IF in > DatatypeLimits.MAX_VALUE_OF_ULINT_WHICH_CAN_BE_HELD_IN_A_UINT THEN
	RETURN;
END_IF

out := ULINT_TO_UINT(in);
TryConvert_ULINT_TO_UINT := TRUE;

END_FUNCTION

// mobject-converters/Converters/ULINT_TO_/TryConvert_ULINT_TO_UDINT
FUNCTION TryConvert_ULINT_TO_UDINT : BOOL
VAR_INPUT
	in : ULINT;
	out : REFERENCE TO UDINT;
END_VAR

IF in > DatatypeLimits.MAX_VALUE_OF_ULINT_WHICH_CAN_BE_HELD_IN_A_UDINT THEN
	RETURN;
END_IF

out := ULINT_TO_UDINT(in);
TryConvert_ULINT_TO_UDINT := TRUE;

END_FUNCTION

// mobject-converters/Converters/ULINT_TO_/TryConvert_ULINT_TO_ULINT
FUNCTION TryConvert_ULINT_TO_ULINT : BOOL
VAR_INPUT
	in : ULINT;
	out : REFERENCE TO ULINT;
END_VAR

out := in;
TryConvert_ULINT_TO_ULINT := TRUE;

END_FUNCTION

// mobject-converters/Converters/ULINT_TO_/TryConvert_ULINT_TO_REAL
FUNCTION TryConvert_ULINT_TO_REAL : BOOL
VAR_INPUT
	in : ULINT;
	out : REFERENCE TO REAL;
END_VAR

out := ULINT_TO_REAL(in);
TryConvert_ULINT_TO_REAL := TRUE;

END_FUNCTION

// mobject-converters/Converters/ULINT_TO_/TryConvert_ULINT_TO_LREAL
FUNCTION TryConvert_ULINT_TO_LREAL : BOOL
VAR_INPUT
	in : ULINT;
	out : REFERENCE TO LREAL;
END_VAR

out := ULINT_TO_LREAL(in);
TryConvert_ULINT_TO_LREAL := TRUE;

END_FUNCTION

// mobject-converters/Converters/ULINT_TO_/TryConvert_ULINT_TO_TIME
FUNCTION TryConvert_ULINT_TO_TIME : BOOL
VAR_INPUT
	in : ULINT;
	out : REFERENCE TO TIME;
END_VAR

IF in > DatatypeLimits.MAX_VALUE_OF_ULINT_WHICH_CAN_BE_HELD_IN_A_TIME THEN
	RETURN;
END_IF

out := ULINT_TO_TIME(in);
TryConvert_ULINT_TO_TIME := TRUE;

END_FUNCTION

// mobject-converters/Converters/ULINT_TO_/TryConvert_ULINT_TO_TOD
FUNCTION TryConvert_ULINT_TO_TOD : BOOL
VAR_INPUT
	in : ULINT;
	out : REFERENCE TO TOD;
END_VAR

IF in > DatatypeLimits.MAX_VALUE_OF_ULINT_WHICH_CAN_BE_HELD_IN_A_TOD THEN
	RETURN;
END_IF

out := ULINT_TO_TOD(in);
TryConvert_ULINT_TO_TOD := TRUE;

END_FUNCTION

// mobject-converters/Converters/ULINT_TO_/TryConvert_ULINT_TO_DT
FUNCTION TryConvert_ULINT_TO_DT : BOOL
VAR_INPUT
	in : ULINT;
	out : REFERENCE TO DT;
END_VAR

IF in > DatatypeLimits.MAX_VALUE_OF_ULINT_WHICH_CAN_BE_HELD_IN_A_DT THEN
	RETURN;
END_IF

out := ULINT_TO_DT(in);
TryConvert_ULINT_TO_DT := TRUE;

END_FUNCTION

// mobject-converters/Converters/ULINT_TO_/TryConvert_ULINT_TO_STRING
FUNCTION TryConvert_ULINT_TO_STRING : BOOL
VAR_INPUT
	in : ULINT;
	out : REFERENCE TO STRING;
END_VAR

out := ULINT_TO_STRING(in);
TryConvert_ULINT_TO_STRING := TRUE;

END_FUNCTION

// mobject-converters/Converters/USINT_TO_/TryConvert_USINT_TO_BOOL
FUNCTION TryConvert_USINT_TO_BOOL : BOOL
VAR_INPUT
	in : USINT;
	out : REFERENCE TO BOOL;
END_VAR

out := USINT_TO_BOOL(in);
TryConvert_USINT_TO_BOOL := TRUE;

END_FUNCTION

// mobject-converters/Converters/USINT_TO_/TryConvert_USINT_TO_BYTE
FUNCTION TryConvert_USINT_TO_BYTE : BOOL
VAR_INPUT
	in : USINT;
	out : REFERENCE TO BYTE;
END_VAR

out := USINT_TO_BYTE(in);
TryConvert_USINT_TO_BYTE := TRUE;

END_FUNCTION

// mobject-converters/Converters/USINT_TO_/TryConvert_USINT_TO_DATE
FUNCTION TryConvert_USINT_TO_DATE : BOOL
VAR_INPUT
	in : USINT;
	out : REFERENCE TO DATE;
END_VAR

out := USINT_TO_DATE(in);
TryConvert_USINT_TO_DATE := TRUE;

END_FUNCTION

// mobject-converters/Converters/USINT_TO_/TryConvert_USINT_TO_Destination
FUNCTION TryConvert_USINT_TO_Destination : BOOL
VAR_INPUT
	in : USINT;
	out : ANY;
END_VAR
VAR
	convertResult : BOOL := FALSE;
	convertAddress : PVOID;
	_BOOL : BOOL;
	_BYTE : BYTE;
	_WORD : WORD;
	_DWORD : DWORD;
	_LWORD : LWORD;
	_SINT : SINT;
	_INT : INT;
	_DINT : DINT;
	_LINT : LINT;
	_USINT : USINT;
	_UINT : UINT;
	_UDINT : UDINT;
	_ULINT : ULINT;
	_REAL : REAL;
	_LREAL : LREAL;
	_TIME : TIME;
	_TOD : TOD;
	_DATE : DATE;
	_DT : DT;
	_STRING : STRING;
END_VAR

CASE out.TypeClass OF
	__SYSTEM.TYPE_CLASS.TYPE_BOOL:
	
	convertResult := TryConvert_USINT_TO_BOOL(in, _BOOL);
	IF convertResult THEN
		convertAddress := ADR(_BOOL);
	END_IF
	
	__SYSTEM.TYPE_CLASS.TYPE_BYTE:
	
	convertResult := TryConvert_USINT_TO_BYTE(in, _BYTE);
	IF convertResult THEN
		convertAddress := ADR(_BYTE);
	END_IF
	
	__SYSTEM.TYPE_CLASS.TYPE_WORD:
	
	convertResult := TryConvert_USINT_TO_WORD(in, _WORD);
	IF convertResult THEN
		convertAddress := ADR(_WORD);
	END_IF
	
	__SYSTEM.TYPE_CLASS.TYPE_DWORD:
	
	convertResult := TryConvert_USINT_TO_DWORD(in, _DWORD);
	IF convertResult THEN
		convertAddress := ADR(_DWORD);
	END_IF
	
	__SYSTEM.TYPE_CLASS.TYPE_LWORD:
	
	convertResult := TryConvert_USINT_TO_LWORD(in, _LWORD);
	IF convertResult THEN
		convertAddress := ADR(_LWORD);
	END_IF
	
	__SYSTEM.TYPE_CLASS.TYPE_SINT:
	
	convertResult := TryConvert_USINT_TO_SINT(in, _SINT);
	IF convertResult THEN
		convertAddress := ADR(_SINT);
	END_IF
	
	__SYSTEM.TYPE_CLASS.TYPE_INT:
	
	convertResult := TryConvert_USINT_TO_INT(in, _INT);
	IF convertResult THEN
		convertAddress := ADR(_INT);
	END_IF
	
	__SYSTEM.TYPE_CLASS.TYPE_DINT:
	
	convertResult := TryConvert_USINT_TO_DINT(in, _DINT);
	IF convertResult THEN
		convertAddress := ADR(_DINT);
	END_IF
	
	__SYSTEM.TYPE_CLASS.TYPE_LINT:
	
	convertResult := TryConvert_USINT_TO_LINT(in, _LINT);
	IF convertResult THEN
		convertAddress := ADR(_LINT);
	END_IF
	
	__SYSTEM.TYPE_CLASS.TYPE_USINT:
	
	convertResult := TryConvert_USINT_TO_USINT(in, _USINT);
	IF convertResult THEN
		convertAddress := ADR(_USINT);
	END_IF
	
	__SYSTEM.TYPE_CLASS.TYPE_UINT:
	
	convertResult := TryConvert_USINT_TO_UINT(in, _UINT);
	IF convertResult THEN
		convertAddress := ADR(_UINT);
	END_IF
	
	__SYSTEM.TYPE_CLASS.TYPE_UDINT:
	
	convertResult := TryConvert_USINT_TO_UDINT(in, _UDINT);
	IF convertResult THEN
		convertAddress := ADR(_UDINT);
	END_IF
	
	__SYSTEM.TYPE_CLASS.TYPE_ULINT:
	
	convertResult := TryConvert_USINT_TO_ULINT(in, _ULINT);
	IF convertResult THEN
		convertAddress := ADR(_ULINT);
	END_IF
	
	__SYSTEM.TYPE_CLASS.TYPE_REAL:
	
	convertResult := TryConvert_USINT_TO_REAL(in, _REAL);
	IF convertResult THEN
		convertAddress := ADR(_REAL);
	END_IF
	
	__SYSTEM.TYPE_CLASS.TYPE_LREAL:
	
	convertResult := TryConvert_USINT_TO_LREAL(in, _LREAL);
	IF convertResult THEN
		convertAddress := ADR(_LREAL);
	END_IF
	
	__SYSTEM.TYPE_CLASS.TYPE_TIME:
	
	convertResult := TryConvert_USINT_TO_TIME(in, _TIME);
	IF convertResult THEN
		convertAddress := ADR(_TIME);
	END_IF
	
	__SYSTEM.TYPE_CLASS.TYPE_TIMEOFDAY:
	
	convertResult := TryConvert_USINT_TO_TOD(in, _TOD);
	IF convertResult THEN
		convertAddress := ADR(_TOD);
	END_IF
	
	__SYSTEM.TYPE_CLASS.TYPE_DATE:
	
	convertResult := TryConvert_USINT_TO_DATE(in, _DATE);
	IF convertResult THEN
		convertAddress := ADR(_DATE);
	END_IF
	
	__SYSTEM.TYPE_CLASS.TYPE_DATEANDTIME:
	
	convertResult := TryConvert_USINT_TO_DT(in, _DT);
	IF convertResult THEN
		convertAddress := ADR(_DT);
	END_IF
	
	__SYSTEM.TYPE_CLASS.TYPE_STRING:
	
	convertResult := TryConvert_USINT_TO_STRING(in, _STRING);
	IF convertResult THEN
		convertAddress := ADR(_STRING);
	END_IF
	
END_CASE

IF convertResult THEN
	memcpy(out.pValue,convertAddress,DINT_TO_UDINT(out.diSize));
END_IF

TryConvert_USINT_TO_Destination := convertResult;

END_FUNCTION

// mobject-converters/Converters/USINT_TO_/TryConvert_USINT_TO_WORD
FUNCTION TryConvert_USINT_TO_WORD : BOOL
VAR_INPUT
	in : USINT;
	out : REFERENCE TO WORD;
END_VAR

out := USINT_TO_WORD(in);
TryConvert_USINT_TO_WORD := TRUE;

END_FUNCTION

// mobject-converters/Converters/USINT_TO_/TryConvert_USINT_TO_DWORD
FUNCTION TryConvert_USINT_TO_DWORD : BOOL
VAR_INPUT
	in : USINT;
	out : REFERENCE TO DWORD;
END_VAR

out := USINT_TO_DWORD(in);
TryConvert_USINT_TO_DWORD := TRUE;

END_FUNCTION

// mobject-converters/Converters/USINT_TO_/TryConvert_USINT_TO_LWORD
FUNCTION TryConvert_USINT_TO_LWORD : BOOL
VAR_INPUT
	in : USINT;
	out : REFERENCE TO LWORD;
END_VAR

out := USINT_TO_LWORD(in);
TryConvert_USINT_TO_LWORD := TRUE;

END_FUNCTION

// mobject-converters/Converters/USINT_TO_/TryConvert_USINT_TO_SINT
FUNCTION TryConvert_USINT_TO_SINT : BOOL
VAR_INPUT
	in : USINT;
	out : REFERENCE TO SINT;
END_VAR

IF in > DatatypeLimits.MAX_VALUE_OF_USINT_WHICH_CAN_BE_HELD_IN_A_SINT THEN
	RETURN;
END_IF

out := USINT_TO_SINT(in);
TryConvert_USINT_TO_SINT := TRUE;

END_FUNCTION

// mobject-converters/Converters/USINT_TO_/TryConvert_USINT_TO_INT
FUNCTION TryConvert_USINT_TO_INT : BOOL
VAR_INPUT
	in : USINT;
	out : REFERENCE TO INT;
END_VAR

out := USINT_TO_INT(in);
TryConvert_USINT_TO_INT := TRUE;

END_FUNCTION

// mobject-converters/Converters/USINT_TO_/TryConvert_USINT_TO_DINT
FUNCTION TryConvert_USINT_TO_DINT : BOOL
VAR_INPUT
	in : USINT;
	out : REFERENCE TO DINT;
END_VAR

out := USINT_TO_DINT(in);
TryConvert_USINT_TO_DINT := TRUE;

END_FUNCTION

// mobject-converters/Converters/USINT_TO_/TryConvert_USINT_TO_LINT
FUNCTION TryConvert_USINT_TO_LINT : BOOL
VAR_INPUT
	in : USINT;
	out : REFERENCE TO LINT;
END_VAR

out := USINT_TO_LINT(in);
TryConvert_USINT_TO_LINT := TRUE;

END_FUNCTION

// mobject-converters/Converters/USINT_TO_/TryConvert_USINT_TO_USINT
FUNCTION TryConvert_USINT_TO_USINT : BOOL
VAR_INPUT
	in : USINT;
	out : REFERENCE TO USINT;
END_VAR

out := in;
TryConvert_USINT_TO_USINT := TRUE;

END_FUNCTION

// mobject-converters/Converters/USINT_TO_/TryConvert_USINT_TO_UINT
FUNCTION TryConvert_USINT_TO_UINT : BOOL
VAR_INPUT
	in : USINT;
	out : REFERENCE TO UINT;
END_VAR

out := USINT_TO_UINT(in);
TryConvert_USINT_TO_UINT := TRUE;

END_FUNCTION

// mobject-converters/Converters/USINT_TO_/TryConvert_USINT_TO_UDINT
FUNCTION TryConvert_USINT_TO_UDINT : BOOL
VAR_INPUT
	in : USINT;
	out : REFERENCE TO UDINT;
END_VAR

out := USINT_TO_UDINT(in);
TryConvert_USINT_TO_UDINT := TRUE;

END_FUNCTION

// mobject-converters/Converters/USINT_TO_/TryConvert_USINT_TO_ULINT
FUNCTION TryConvert_USINT_TO_ULINT : BOOL
VAR_INPUT
	in : USINT;
	out : REFERENCE TO ULINT;
END_VAR

out := USINT_TO_ULINT(in);
TryConvert_USINT_TO_ULINT := TRUE;

END_FUNCTION

// mobject-converters/Converters/USINT_TO_/TryConvert_USINT_TO_REAL
FUNCTION TryConvert_USINT_TO_REAL : BOOL
VAR_INPUT
	in : USINT;
	out : REFERENCE TO REAL;
END_VAR

out := USINT_TO_REAL(in);
TryConvert_USINT_TO_REAL := TRUE;

END_FUNCTION

// mobject-converters/Converters/USINT_TO_/TryConvert_USINT_TO_LREAL
FUNCTION TryConvert_USINT_TO_LREAL : BOOL
VAR_INPUT
	in : USINT;
	out : REFERENCE TO LREAL;
END_VAR

out := USINT_TO_LREAL(in);
TryConvert_USINT_TO_LREAL := TRUE;

END_FUNCTION

// mobject-converters/Converters/USINT_TO_/TryConvert_USINT_TO_TIME
FUNCTION TryConvert_USINT_TO_TIME : BOOL
VAR_INPUT
	in : USINT;
	out : REFERENCE TO TIME;
END_VAR

out := USINT_TO_TIME(in);
TryConvert_USINT_TO_TIME := TRUE;

END_FUNCTION

// mobject-converters/Converters/USINT_TO_/TryConvert_USINT_TO_TOD
FUNCTION TryConvert_USINT_TO_TOD : BOOL
VAR_INPUT
	in : USINT;
	out : REFERENCE TO TOD;
END_VAR

out := USINT_TO_TOD(in);
TryConvert_USINT_TO_TOD := TRUE;

END_FUNCTION

// mobject-converters/Converters/USINT_TO_/TryConvert_USINT_TO_DT
FUNCTION TryConvert_USINT_TO_DT : BOOL
VAR_INPUT
	in : USINT;
	out : REFERENCE TO DT;
END_VAR

out := USINT_TO_DT(in);
TryConvert_USINT_TO_DT := TRUE;

END_FUNCTION

// mobject-converters/Converters/USINT_TO_/TryConvert_USINT_TO_STRING
FUNCTION TryConvert_USINT_TO_STRING : BOOL
VAR_INPUT
	in : USINT;
	out : REFERENCE TO STRING;
END_VAR

out := USINT_TO_STRING(in);
TryConvert_USINT_TO_STRING := TRUE;

END_FUNCTION

// mobject-converters/Converters/WORD_TO_/TryConvert_WORD_TO_BOOL
FUNCTION TryConvert_WORD_TO_BOOL : BOOL
VAR_INPUT
	in : WORD;
	out : REFERENCE TO BOOL;
END_VAR

out := WORD_TO_BOOL(in);
TryConvert_WORD_TO_BOOL := TRUE;

END_FUNCTION

// mobject-converters/Converters/WORD_TO_/TryConvert_WORD_TO_BYTE
FUNCTION TryConvert_WORD_TO_BYTE : BOOL
VAR_INPUT
	in : WORD;
	out : REFERENCE TO BYTE;
END_VAR

IF in > DatatypeLimits.MAX_VALUE_OF_WORD_WHICH_CAN_BE_HELD_IN_A_BYTE THEN
	RETURN;
END_IF

out := WORD_TO_BYTE(in);
TryConvert_WORD_TO_BYTE := TRUE;

END_FUNCTION

// mobject-converters/Converters/WORD_TO_/TryConvert_WORD_TO_DATE
FUNCTION TryConvert_WORD_TO_DATE : BOOL
VAR_INPUT
	in : WORD;
	out : REFERENCE TO DATE;
END_VAR

out := WORD_TO_DATE(in);
TryConvert_WORD_TO_DATE := TRUE;

END_FUNCTION

// mobject-converters/Converters/WORD_TO_/TryConvert_WORD_TO_Destination
FUNCTION TryConvert_WORD_TO_Destination : BOOL
VAR_INPUT
	in : WORD;
	out : ANY;
END_VAR
VAR
	convertResult : BOOL := FALSE;
	convertAddress : PVOID;
	_BOOL : BOOL;
	_BYTE : BYTE;
	_WORD : WORD;
	_DWORD : DWORD;
	_LWORD : LWORD;
	_SINT : SINT;
	_INT : INT;
	_DINT : DINT;
	_LINT : LINT;
	_USINT : USINT;
	_UINT : UINT;
	_UDINT : UDINT;
	_ULINT : ULINT;
	_REAL : REAL;
	_LREAL : LREAL;
	_TIME : TIME;
	_TOD : TOD;
	_DATE : DATE;
	_DT : DT;
	_STRING : STRING;
END_VAR

CASE out.TypeClass OF
	__SYSTEM.TYPE_CLASS.TYPE_BOOL:
	
	convertResult := TryConvert_WORD_TO_BOOL(in, _BOOL);
	IF convertResult THEN
		convertAddress := ADR(_BOOL);
	END_IF
	
	__SYSTEM.TYPE_CLASS.TYPE_BYTE:
	
	convertResult := TryConvert_WORD_TO_BYTE(in, _BYTE);
	IF convertResult THEN
		convertAddress := ADR(_BYTE);
	END_IF
	
	__SYSTEM.TYPE_CLASS.TYPE_WORD:
	
	convertResult := TryConvert_WORD_TO_WORD(in, _WORD);
	IF convertResult THEN
		convertAddress := ADR(_WORD);
	END_IF
	
	__SYSTEM.TYPE_CLASS.TYPE_DWORD:
	
	convertResult := TryConvert_WORD_TO_DWORD(in, _DWORD);
	IF convertResult THEN
		convertAddress := ADR(_DWORD);
	END_IF
	
	__SYSTEM.TYPE_CLASS.TYPE_LWORD:
	
	convertResult := TryConvert_WORD_TO_LWORD(in, _LWORD);
	IF convertResult THEN
		convertAddress := ADR(_LWORD);
	END_IF
	
	__SYSTEM.TYPE_CLASS.TYPE_SINT:
	
	convertResult := TryConvert_WORD_TO_SINT(in, _SINT);
	IF convertResult THEN
		convertAddress := ADR(_SINT);
	END_IF
	
	__SYSTEM.TYPE_CLASS.TYPE_INT:
	
	convertResult := TryConvert_WORD_TO_INT(in, _INT);
	IF convertResult THEN
		convertAddress := ADR(_INT);
	END_IF
	
	__SYSTEM.TYPE_CLASS.TYPE_DINT:
	
	convertResult := TryConvert_WORD_TO_DINT(in, _DINT);
	IF convertResult THEN
		convertAddress := ADR(_DINT);
	END_IF
	
	__SYSTEM.TYPE_CLASS.TYPE_LINT:
	
	convertResult := TryConvert_WORD_TO_LINT(in, _LINT);
	IF convertResult THEN
		convertAddress := ADR(_LINT);
	END_IF
	
	__SYSTEM.TYPE_CLASS.TYPE_USINT:
	
	convertResult := TryConvert_WORD_TO_USINT(in, _USINT);
	IF convertResult THEN
		convertAddress := ADR(_USINT);
	END_IF
	
	__SYSTEM.TYPE_CLASS.TYPE_UINT:
	
	convertResult := TryConvert_WORD_TO_UINT(in, _UINT);
	IF convertResult THEN
		convertAddress := ADR(_UINT);
	END_IF
	
	__SYSTEM.TYPE_CLASS.TYPE_UDINT:
	
	convertResult := TryConvert_WORD_TO_UDINT(in, _UDINT);
	IF convertResult THEN
		convertAddress := ADR(_UDINT);
	END_IF
	
	__SYSTEM.TYPE_CLASS.TYPE_ULINT:
	
	convertResult := TryConvert_WORD_TO_ULINT(in, _ULINT);
	IF convertResult THEN
		convertAddress := ADR(_ULINT);
	END_IF
	
	__SYSTEM.TYPE_CLASS.TYPE_REAL:
	
	convertResult := TryConvert_WORD_TO_REAL(in, _REAL);
	IF convertResult THEN
		convertAddress := ADR(_REAL);
	END_IF
	
	__SYSTEM.TYPE_CLASS.TYPE_LREAL:
	
	convertResult := TryConvert_WORD_TO_LREAL(in, _LREAL);
	IF convertResult THEN
		convertAddress := ADR(_LREAL);
	END_IF
	
	__SYSTEM.TYPE_CLASS.TYPE_TIME:
	
	convertResult := TryConvert_WORD_TO_TIME(in, _TIME);
	IF convertResult THEN
		convertAddress := ADR(_TIME);
	END_IF
	
	__SYSTEM.TYPE_CLASS.TYPE_TIMEOFDAY:
	
	convertResult := TryConvert_WORD_TO_TOD(in, _TOD);
	IF convertResult THEN
		convertAddress := ADR(_TOD);
	END_IF
	
	__SYSTEM.TYPE_CLASS.TYPE_DATE:
	
	convertResult := TryConvert_WORD_TO_DATE(in, _DATE);
	IF convertResult THEN
		convertAddress := ADR(_DATE);
	END_IF
	
	__SYSTEM.TYPE_CLASS.TYPE_DATEANDTIME:
	
	convertResult := TryConvert_WORD_TO_DT(in, _DT);
	IF convertResult THEN
		convertAddress := ADR(_DT);
	END_IF
	
	__SYSTEM.TYPE_CLASS.TYPE_STRING:
	
	convertResult := TryConvert_WORD_TO_STRING(in, _STRING);
	IF convertResult THEN
		convertAddress := ADR(_STRING);
	END_IF
	
END_CASE

IF convertResult THEN
	memcpy(out.pValue,convertAddress,DINT_TO_UDINT(out.diSize));
END_IF

TryConvert_WORD_TO_Destination := convertResult;

END_FUNCTION

// mobject-converters/Converters/WORD_TO_/TryConvert_WORD_TO_WORD
FUNCTION TryConvert_WORD_TO_WORD : BOOL
VAR_INPUT
	in : WORD;
	out : REFERENCE TO WORD;
END_VAR

out := in;
TryConvert_WORD_TO_WORD := TRUE;

END_FUNCTION

// mobject-converters/Converters/WORD_TO_/TryConvert_WORD_TO_DWORD
FUNCTION TryConvert_WORD_TO_DWORD : BOOL
VAR_INPUT
	in : WORD;
	out : REFERENCE TO DWORD;
END_VAR

out := WORD_TO_DWORD(in);
TryConvert_WORD_TO_DWORD := TRUE;

END_FUNCTION

// mobject-converters/Converters/WORD_TO_/TryConvert_WORD_TO_LWORD
FUNCTION TryConvert_WORD_TO_LWORD : BOOL
VAR_INPUT
	in : WORD;
	out : REFERENCE TO LWORD;
END_VAR

out := WORD_TO_LWORD(in);
TryConvert_WORD_TO_LWORD := TRUE;

END_FUNCTION

// mobject-converters/Converters/WORD_TO_/TryConvert_WORD_TO_SINT
FUNCTION TryConvert_WORD_TO_SINT : BOOL
VAR_INPUT
	in : WORD;
	out : REFERENCE TO SINT;
END_VAR

IF in > DatatypeLimits.MAX_VALUE_OF_WORD_WHICH_CAN_BE_HELD_IN_A_SINT THEN
	RETURN;
END_IF

out := WORD_TO_SINT(in);
TryConvert_WORD_TO_SINT := TRUE;

END_FUNCTION

// mobject-converters/Converters/WORD_TO_/TryConvert_WORD_TO_INT
FUNCTION TryConvert_WORD_TO_INT : BOOL
VAR_INPUT
	in : WORD;
	out : REFERENCE TO INT;
END_VAR

IF in > DatatypeLimits.MAX_VALUE_OF_WORD_WHICH_CAN_BE_HELD_IN_A_INT THEN
	RETURN;
END_IF

out := WORD_TO_INT(in);
TryConvert_WORD_TO_INT := TRUE;

END_FUNCTION

// mobject-converters/Converters/WORD_TO_/TryConvert_WORD_TO_DINT
FUNCTION TryConvert_WORD_TO_DINT : BOOL
VAR_INPUT
	in : WORD;
	out : REFERENCE TO DINT;
END_VAR

out := WORD_TO_DINT(in);
TryConvert_WORD_TO_DINT := TRUE;

END_FUNCTION

// mobject-converters/Converters/WORD_TO_/TryConvert_WORD_TO_LINT
FUNCTION TryConvert_WORD_TO_LINT : BOOL
VAR_INPUT
	in : WORD;
	out : REFERENCE TO LINT;
END_VAR

out := WORD_TO_LINT(in);
TryConvert_WORD_TO_LINT := TRUE;

END_FUNCTION

// mobject-converters/Converters/WORD_TO_/TryConvert_WORD_TO_USINT
FUNCTION TryConvert_WORD_TO_USINT : BOOL
VAR_INPUT
	in : WORD;
	out : REFERENCE TO USINT;
END_VAR

IF in > DatatypeLimits.MAX_VALUE_OF_WORD_WHICH_CAN_BE_HELD_IN_A_USINT THEN
	RETURN;
END_IF

out := WORD_TO_USINT(in);
TryConvert_WORD_TO_USINT := TRUE;

END_FUNCTION

// mobject-converters/Converters/WORD_TO_/TryConvert_WORD_TO_UINT
FUNCTION TryConvert_WORD_TO_UINT : BOOL
VAR_INPUT
	in : WORD;
	out : REFERENCE TO UINT;
END_VAR

out := WORD_TO_UINT(in);
TryConvert_WORD_TO_UINT := TRUE;

END_FUNCTION

// mobject-converters/Converters/WORD_TO_/TryConvert_WORD_TO_UDINT
FUNCTION TryConvert_WORD_TO_UDINT : BOOL
VAR_INPUT
	in : WORD;
	out : REFERENCE TO UDINT;
END_VAR

out := WORD_TO_UDINT(in);
TryConvert_WORD_TO_UDINT := TRUE;

END_FUNCTION

// mobject-converters/Converters/WORD_TO_/TryConvert_WORD_TO_ULINT
FUNCTION TryConvert_WORD_TO_ULINT : BOOL
VAR_INPUT
	in : WORD;
	out : REFERENCE TO ULINT;
END_VAR

out := WORD_TO_ULINT(in);
TryConvert_WORD_TO_ULINT := TRUE;

END_FUNCTION

// mobject-converters/Converters/WORD_TO_/TryConvert_WORD_TO_REAL
FUNCTION TryConvert_WORD_TO_REAL : BOOL
VAR_INPUT
	in : WORD;
	out : REFERENCE TO REAL;
END_VAR

out := WORD_TO_REAL(in);
TryConvert_WORD_TO_REAL := TRUE;

END_FUNCTION

// mobject-converters/Converters/WORD_TO_/TryConvert_WORD_TO_LREAL
FUNCTION TryConvert_WORD_TO_LREAL : BOOL
VAR_INPUT
	in : WORD;
	out : REFERENCE TO LREAL;
END_VAR

out := WORD_TO_LREAL(in);
TryConvert_WORD_TO_LREAL := TRUE;

END_FUNCTION

// mobject-converters/Converters/WORD_TO_/TryConvert_WORD_TO_TIME
FUNCTION TryConvert_WORD_TO_TIME : BOOL
VAR_INPUT
	in : WORD;
	out : REFERENCE TO TIME;
END_VAR

out := WORD_TO_TIME(in);
TryConvert_WORD_TO_TIME := TRUE;

END_FUNCTION

// mobject-converters/Converters/WORD_TO_/TryConvert_WORD_TO_TOD
FUNCTION TryConvert_WORD_TO_TOD : BOOL
VAR_INPUT
	in : WORD;
	out : REFERENCE TO TOD;
END_VAR

out := WORD_TO_TOD(in);
TryConvert_WORD_TO_TOD := TRUE;

END_FUNCTION

// mobject-converters/Converters/WORD_TO_/TryConvert_WORD_TO_DT
FUNCTION TryConvert_WORD_TO_DT : BOOL
VAR_INPUT
	in : WORD;
	out : REFERENCE TO DT;
END_VAR

out := WORD_TO_DT(in);
TryConvert_WORD_TO_DT := TRUE;

END_FUNCTION

// mobject-converters/Converters/WORD_TO_/TryConvert_WORD_TO_STRING
FUNCTION TryConvert_WORD_TO_STRING : BOOL
VAR_INPUT
	in : WORD;
	out : REFERENCE TO STRING;
END_VAR

out := WORD_TO_STRING(in);
TryConvert_WORD_TO_STRING := TRUE;

END_FUNCTION

// mobject-converters/Converters/TryConvert_Source_TO_Destination
{attribute 'linkalways'} 
FUNCTION TryConvert_Source_TO_Destination : BOOL
VAR_INPUT
	in : ANY;
	out : ANY;
END_VAR
VAR
	_BOOL : BOOL;
	_BYTE : BYTE;
	_WORD : WORD;
	_DWORD : DWORD;
	_LWORD : LWORD;
	_SINT : SINT;
	_INT : INT;
	_DINT : DINT;
	_LINT : LINT;
	_USINT : USINT;
	_UINT : UINT;
	_UDINT : UDINT;
	_ULINT : ULINT;
	_REAL : REAL;
	_LREAL : LREAL;
	_TIME : TIME;
	_TOD : TOD;
	_DATE : DATE;
	_DT : DT;
	_STRING : STRING;
	convertResult : BOOL := FALSE;
END_VAR

CASE in.TypeClass OF

	__SYSTEM.TYPE_CLASS.TYPE_BOOL :
		memcpy(ADR(_BOOL),in.pValue,DINT_TO_UDINT(in.diSize));
		convertResult := TryConvert_BOOL_To_Destination(_BOOL, out);
		
	__SYSTEM.TYPE_CLASS.TYPE_BYTE :
		memcpy(ADR(_BYTE),in.pValue,DINT_TO_UDINT(in.diSize));
		convertResult := TryConvert_BYTE_To_Destination(_BYTE, out);
		
	__SYSTEM.TYPE_CLASS.TYPE_WORD :
		memcpy(ADR(_WORD),in.pValue,DINT_TO_UDINT(in.diSize));
		convertResult := TryConvert_WORD_To_Destination(_WORD, out);
		
	__SYSTEM.TYPE_CLASS.TYPE_DWORD :
		memcpy(ADR(_DWORD),in.pValue,DINT_TO_UDINT(in.diSize));
		convertResult := TryConvert_DWORD_To_Destination(_DWORD, out);
		
	__SYSTEM.TYPE_CLASS.TYPE_LWORD :
		memcpy(ADR(_LWORD),in.pValue,DINT_TO_UDINT(in.diSize));
		convertResult := TryConvert_LWORD_To_Destination(_LWORD, out);
		
	__SYSTEM.TYPE_CLASS.TYPE_SINT :
		memcpy(ADR(_SINT),in.pValue,DINT_TO_UDINT(in.diSize));
		convertResult := TryConvert_SINT_To_Destination(_SINT, out);
		
	__SYSTEM.TYPE_CLASS.TYPE_INT :
		memcpy(ADR(_INT),in.pValue,DINT_TO_UDINT(in.diSize));
		convertResult := TryConvert_INT_To_Destination(_INT, out);
		
	__SYSTEM.TYPE_CLASS.TYPE_DINT :
		memcpy(ADR(_DINT),in.pValue,DINT_TO_UDINT(in.diSize));
		convertResult := TryConvert_DINT_To_Destination(_DINT, out);
		
	__SYSTEM.TYPE_CLASS.TYPE_LINT :
		memcpy(ADR(_LINT),in.pValue,DINT_TO_UDINT(in.diSize));
		convertResult := TryConvert_LINT_To_Destination(_LINT, out);
		
	__SYSTEM.TYPE_CLASS.TYPE_USINT :
		memcpy(ADR(_USINT),in.pValue,DINT_TO_UDINT(in.diSize));
		convertResult := TryConvert_USINT_To_Destination(_USINT, out);
		
	__SYSTEM.TYPE_CLASS.TYPE_UINT :
		memcpy(ADR(_UINT),in.pValue,DINT_TO_UDINT(in.diSize));
		convertResult := TryConvert_UINT_To_Destination(_UINT, out);
		
	__SYSTEM.TYPE_CLASS.TYPE_UDINT :
		memcpy(ADR(_UDINT),in.pValue,DINT_TO_UDINT(in.diSize));
		convertResult := TryConvert_UDINT_To_Destination(_UDINT, out);
		
	__SYSTEM.TYPE_CLASS.TYPE_ULINT :
		memcpy(ADR(_ULINT),in.pValue,DINT_TO_UDINT(in.diSize));
		convertResult := TryConvert_ULINT_To_Destination(_ULINT, out);
		
	__SYSTEM.TYPE_CLASS.TYPE_REAL :
		memcpy(ADR(_REAL),in.pValue,DINT_TO_UDINT(in.diSize));
		convertResult := TryConvert_REAL_To_Destination(_REAL, out);
		
	__SYSTEM.TYPE_CLASS.TYPE_LREAL :
		memcpy(ADR(_LREAL),in.pValue,DINT_TO_UDINT(in.diSize));
		convertResult := TryConvert_LREAL_To_Destination(_LREAL, out);
		
	__SYSTEM.TYPE_CLASS.TYPE_TIME :
		memcpy(ADR(_TIME),in.pValue,DINT_TO_UDINT(in.diSize));
		convertResult := TryConvert_TIME_To_Destination(_TIME, out);
		
	__SYSTEM.TYPE_CLASS.TYPE_TIMEOFDAY :
		memcpy(ADR(_TOD),in.pValue,DINT_TO_UDINT(in.diSize));
		convertResult := TryConvert_TOD_To_Destination(_TOD, out);
		
	__SYSTEM.TYPE_CLASS.TYPE_DATE :
		memcpy(ADR(_DATE),in.pValue,DINT_TO_UDINT(in.diSize));
		convertResult := TryConvert_DATE_To_Destination(_DATE, out);
		
	__SYSTEM.TYPE_CLASS.TYPE_DATEANDTIME :
		memcpy(ADR(_DT),in.pValue,DINT_TO_UDINT(in.diSize));
		convertResult := TryConvert_DT_To_Destination(_DT, out);
		
	__SYSTEM.TYPE_CLASS.TYPE_STRING :
		memcpy(ADR(_STRING),in.pValue,DINT_TO_UDINT(in.diSize));
		convertResult := TryConvert_STRING_To_Destination(_STRING, out);
		
	END_CASE
TryConvert_Source_TO_Destination  := convertResult;

END_FUNCTION

// mobject-datatypes/_Internal/Datatype/AliasDatatypeBase
{attribute 'linkalways'} 
{attribute 'no_explicit_call' := 'This FB is a CLASS and must be accessed using methods or properties'}
{attribute 'enable_dynamic_creation'}
FUNCTION_BLOCK ABSTRACT AliasDatatypeBase EXTENDS UserDefinedDatatypeBase IMPLEMENTS I_AliasDatatype
VAR
	_baseDatatype : I_Datatype;
END_VAR

METHOD PROTECTED AddBaseDatatype
VAR_INPUT
	BaseType : I_Datatype;
END_VAR
_baseDatatype := BaseType;
END_METHOD

METHOD PROTECTED OnSerializeTypeWith
VAR_INPUT
	Serializer : I_Serializer;
END_VAR
SUPER^.OnSerializeTypeWith(Serializer);
Serializer.AddKey('baseDatatype');
_baseDatatype.SerializeTypeWith(Serializer);
END_METHOD

PROPERTY PUBLIC BaseDatatype : I_Datatype
GET
BaseDatatype := _baseDatatype;
END_GET
END_PROPERTY

METHOD PUBLIC SerializeWith
VAR_INPUT
	Serializer : I_Serializer;
END_VAR
_baseDatatype.SerializeWith(Serializer);
END_METHOD

METHOD TryDeserializeFrom : BOOL
VAR_INPUT
	Deserializer : I_Deserializer;
	Feedback : I_DeserializerFeedback;
END_VAR
TryDeserializeFrom := _baseDatatype.TryDeserializeFrom(Deserializer, Feedback);
END_METHOD

METHOD PUBLIC TryResolveAsAliasDatatype : BOOL
VAR_INPUT
	Destination : REFERENCE TO I_AliasDatatype;
END_VAR
Destination := THIS^;
TryResolveAsAliasDatatype := TRUE;
END_METHOD

PROPERTY PUBLIC TypeName : T_MAXSTRING
GET
TypeName := 'ALIAS';
END_GET
END_PROPERTY

END_FUNCTION_BLOCK

// mobject-datatypes/_Internal/Datatype/UserDefinedDatatypeBase
{attribute 'linkalways'} 
{attribute 'no_explicit_call' := 'This FB is a CLASS and must be accessed using methods or properties'}
{attribute 'enable_dynamic_creation'}
FUNCTION_BLOCK ABSTRACT UserDefinedDatatypeBase EXTENDS DatatypeBase IMPLEMENTS I_UserDefinedDatatype
VAR
END_VAR

METHOD PROTECTED OnSerializeTypeWith
VAR_INPUT
	Serializer : I_Serializer;
END_VAR
SUPER^.OnSerializeTypeWith(Serializer);
Serializer.AddKeyString('identifier',Identifier);
END_METHOD

PROPERTY PUBLIC ABSTRACT Identifier : T_MAXSTRING
GET
END_GET
END_PROPERTY

PROPERTY PUBLIC IsUserDefined : BOOL
GET
IsUserDefined := TRUE;
END_GET
END_PROPERTY

METHOD PUBLIC TryCopyFrom : BOOL
VAR_INPUT
	Source : I_Datatype;
END_VAR
VAR
	sourceAsUdt : I_UserDefinedDatatype;
END_VAR
IF NOT __QUERYINTERFACE(Source, sourceAsUdt) THEN
	RETURN;
END_IF

IF sourceAsUdt.Identifier <> Identifier THEN
	RETURN;
END_IF

TryCopyFrom := SUPER^.TryCopyFrom(Source);
END_METHOD

METHOD PUBLIC TryResolveAsUserDefinedDatatype : BOOL
VAR_INPUT
	Destination : REFERENCE TO I_UserDefinedDatatype;
END_VAR
Destination := THIS^;
TryResolveAsUserDefinedDatatype := TRUE;
END_METHOD

END_FUNCTION_BLOCK

// mobject-datatypes/_Internal/Datatype/ArrayDatatypeBase
{attribute 'linkalways'} 
{attribute 'no_explicit_call' := 'This FB is a CLASS and must be accessed using methods or properties'}
{attribute 'enable_dynamic_creation'}
FUNCTION_BLOCK ABSTRACT ArrayDatatypeBase EXTENDS UserDefinedDatatypeBase IMPLEMENTS I_ArrayDatatype
VAR
END_VAR

METHOD PRIVATE CreateEnumError : I_Error
VAR_INPUT
	Enum : T_MAXSTRING;
END_VAR
VAR
	pError : POINTER TO UnknownEnumerationError;
END_VAR
pError := __NEW(UnknownEnumerationError(EnumString := Enum));
CreateEnumError := pError^;
END_METHOD

METHOD PRIVATE SerializeBaseType
VAR_INPUT
	Serializer : I_Serializer;
END_VAR
IF BaseDatatype = 0 THEN
	RETURN;
END_IF

Serializer.AddKey('baseType');
BaseDatatype.SerializeTypeWith(Serializer);
END_METHOD

METHOD PROTECTED ABSTRACT OnSerializeArrayValues
VAR_INPUT
	Serializer : I_Serializer;
END_VAR
END_METHOD

METHOD PROTECTED OnSerializeTypeWith
VAR_INPUT
	Serializer : I_Serializer;
END_VAR
SUPER^.OnSerializeTypeWith(Serializer);
SerializeBaseType(Serializer);
END_METHOD

METHOD PROTECTED ABSTRACT TryDeserializeArrayValues : BOOL
VAR_INPUT
	Deserializer : I_Deserializer;
	Feedback : I_DeserializerFeedback;
END_VAR
END_METHOD

PROPERTY PUBLIC ABSTRACT BaseDatatype : I_Datatype
GET
END_GET
END_PROPERTY

METHOD PUBLIC ABSTRACT GetElementAsDatatypeByIndex : I_Datatype
VAR_INPUT
	Index : DINT;
END_VAR
END_METHOD

PROPERTY PUBLIC Identifier : T_MAXSTRING
GET
VAR
	baseTypeAsUdt : I_UserDefinedDatatype;
END_VAR
Identifier := Concat('ARRAY [', DINT_TO_STRING(LowerBound));
Identifier := Concat(Identifier,'..');
Identifier := Concat(Identifier, DINT_TO_STRING(UpperBound));
Identifier := Concat(Identifier, '] OF ');

IF BaseDatatype.TryResolveAsUserDefinedDatatype(baseTypeAsUdt) THEN
	Identifier := Concat(Identifier, baseTypeAsUdt.Identifier);
ELSE
	Identifier := Concat(Identifier, BaseDatatype.TypeName);
END_IF
END_GET
END_PROPERTY

PROPERTY PUBLIC Length : UDINT
GET
Length := ABS(UpperBound - LowerBound) + 1;
END_GET
END_PROPERTY

PROPERTY PUBLIC ABSTRACT LowerBound : DINT
GET
END_GET
END_PROPERTY

METHOD PUBLIC SerializeWith
VAR_INPUT
	Serializer : I_Serializer;
END_VAR
Serializer.StartArray();
OnSerializeArrayValues(Serializer);
Serializer.EndArray();
END_METHOD

METHOD TryDeserializeFrom : BOOL
VAR_INPUT
	Deserializer : I_Deserializer;
	Feedback : I_DeserializerFeedback;
END_VAR
TryDeserializeFrom := TryDeserializeArrayValues(Deserializer, Feedback);
END_METHOD

METHOD PUBLIC TryResolveAsArrayDatatype : BOOL
VAR_INPUT
	Destination : REFERENCE TO I_ArrayDatatype;
END_VAR
Destination := THIS^;
TryResolveAsArrayDatatype := TRUE;
END_METHOD

PROPERTY PUBLIC TypeName : T_MAXSTRING
GET
TypeName := 'ARRAY';
END_GET
END_PROPERTY

PROPERTY PUBLIC ABSTRACT UpperBound : DINT
GET
END_GET
END_PROPERTY

END_FUNCTION_BLOCK

// mobject-datatypes/_Internal/Errors/UnknownEnumerationError
{attribute 'linkalways'} 
{attribute 'no_explicit_call' := 'This FB is a CLASS and must be accessed using methods or properties'}
{attribute 'enable_dynamic_creation'}
FUNCTION_BLOCK UnknownEnumerationError EXTENDS Error
VAR
	enumString : T_MAXSTRING;
END_VAR

METHOD FB_init : BOOL
VAR_INPUT
	bInitRetains : BOOL; // if TRUE, the retain variables are initialized (warm start / cold start)
	bInCopyCode : BOOL;  // if TRUE, the instance afterwards gets moved into the copy code (online change)
	EnumString : T_MAXSTRING;
END_VAR
THIS^.enumString := EnumString;
END_METHOD

PROPERTY PUBLIC ErrorType : T_MAXSTRING
GET
ErrorType := 'UNKNOWN_ENUMERATION_ERROR';
END_GET
END_PROPERTY

PROPERTY PUBLIC Message : T_MAXSTRING
GET
Message := CONCAT('Unknown Enumeration : ', enumString);
END_GET
END_PROPERTY

END_FUNCTION_BLOCK

// mobject-datatypes/_Internal/Datatype/EnumDatatypeBase
{attribute 'linkalways'} 
{attribute 'no_explicit_call' := 'This FB is a CLASS and must be accessed using methods or properties'}
{attribute 'enable_dynamic_creation'}
FUNCTION_BLOCK ABSTRACT EnumDatatypeBase EXTENDS UserDefinedDatatypeBase IMPLEMENTS I_EnumDatatype
VAR
	_baseDatatype : I_Datatype;
	enumerations : OrderedDictionary;
END_VAR

METHOD PRIVATE CreateEnumError : I_Error
VAR_INPUT
	Enum : T_MAXSTRING;
END_VAR
VAR
	pError : POINTER TO UnknownEnumerationError;
END_VAR
pError := __NEW(UnknownEnumerationError(EnumString := Enum));
CreateEnumError := pError^;
END_METHOD

METHOD PRIVATE SerializeBaseType
VAR_INPUT
	Serializer : I_Serializer;
END_VAR
IF _baseDatatype = 0 THEN
	RETURN;
END_IF

Serializer.AddKey('baseType');
_baseDatatype.SerializeTypeWith(Serializer);
END_METHOD

METHOD PRIVATE SerializeEnums
VAR_INPUT
	Serializer : I_Serializer;
END_VAR
VAR
	enumerator : I_KeyValueForwardEnumerator;
END_VAR
Serializer.AddKey('enumerations');
Serializer.StartArray();

enumerator := enumerations.GetKeyValueEnumerator();

WHILE enumerator.MoveNext() DO
	Serializer.AddString(enumerator.Key);
END_WHILE

enumerator.Dispose();

Serializer.EndArray();
END_METHOD

METHOD PROTECTED AddBaseDatatype
VAR_INPUT
	BaseType : I_Datatype;
END_VAR
_baseDatatype := BaseType;
END_METHOD

METHOD PROTECTED AddEnumeration
VAR_INPUT
	Enumeration : T_MAXSTRING;
	Value : ANY;
END_VAR
enumerations.AddOrUpdate(Enumeration, Value);
END_METHOD

METHOD ABSTRACT IsEnumeratorValueEqual : BOOL
VAR_INPUT
	Enumerator : I_KeyValueForwardEnumerator;
END_VAR
END_METHOD

METHOD PROTECTED OnSerializeTypeWith
VAR_INPUT
	Serializer : I_Serializer;
END_VAR
SUPER^.OnSerializeTypeWith(Serializer);
SerializeEnums(Serializer);
SerializeBaseType(Serializer);
END_METHOD

PROPERTY PUBLIC BaseDatatype : I_Datatype
GET
BaseDatatype := _baseDatatype;
END_GET
END_PROPERTY

METHOD PUBLIC SerializeWith
VAR_INPUT
	Serializer : I_Serializer;
END_VAR
VAR
	returnKey : T_MAXSTRING;
	enumerator : I_KeyValueForwardEnumerator;
END_VAR
enumerator := enumerations.GetKeyValueEnumerator();
returnKey := 'UNDEFINED';

WHILE (enumerator.MoveNext()) DO
	
	IF IsEnumeratorValueEqual(enumerator) THEN
		returnKey := enumerator.key;
		EXIT;
	END_IF

END_WHILE

Serializer.AddString(returnKey);
enumerator.Dispose();
END_METHOD

METHOD TryDeserializeFrom : BOOL
VAR_INPUT
	Deserializer : I_Deserializer;
	Feedback : I_DeserializerFeedback;
END_VAR
VAR
	key : T_MAXSTRING;
	error : I_Error;
END_VAR
IF NOT Deserializer.TryGetString(key, Feedback) THEN
	RETURN;
END_IF

IF NOT enumerations.TryGetValueTo(key, Address, Size) THEN
	error := CreateEnumError(key);
	Feedback.LogError(error);
	RETURN;
END_IF

TryDeserializeFrom := TRUE;
END_METHOD

METHOD PUBLIC TryResolveAsEnumDatatype : BOOL
VAR_INPUT
	Destination : REFERENCE TO I_EnumDatatype;
END_VAR
Destination := THIS^;
TryResolveAsEnumDatatype := TRUE;
END_METHOD

PROPERTY PUBLIC TypeName : T_MAXSTRING
GET
TypeName := 'ENUM';
END_GET
END_PROPERTY

END_FUNCTION_BLOCK

// mobject-datatypes/_Internal/Datatype/InterfaceDatatypeBase
{attribute 'linkalways'} 
{attribute 'no_explicit_call' := 'This FB is a CLASS and must be accessed using methods or properties'}
{attribute 'enable_dynamic_creation'}
FUNCTION_BLOCK ABSTRACT InterfaceDatatypeBase EXTENDS DatatypeBase IMPLEMENTS I_InterfaceDatatype
VAR
END_VAR

METHOD PROTECTED OnSerializeTypeWith
VAR_INPUT
	Serializer : I_Serializer;
END_VAR
SUPER^.OnSerializeTypeWith(Serializer);
Serializer.AddKeyString('identifier',Identifier);
END_METHOD

PROPERTY PUBLIC ABSTRACT Identifier : T_MAXSTRING
GET
END_GET
END_PROPERTY

PROPERTY PUBLIC IsUserDefined : BOOL
GET
IsUserDefined := FALSE;
END_GET
END_PROPERTY

METHOD PUBLIC TryCopyFrom : BOOL
VAR_INPUT
	Source : I_Datatype;
END_VAR
VAR
	sourceAsInterface : I_InterfaceDatatype;
END_VAR
IF NOT __QUERYINTERFACE(Source, sourceAsInterface) THEN
	RETURN;
END_IF

IF sourceAsInterface.Identifier <> Identifier THEN
	RETURN;
END_IF

TryCopyFrom := SUPER^.TryCopyFrom(Source);
END_METHOD

METHOD PUBLIC TryResolveAsInterfaceDatatype : BOOL
VAR_INPUT
	Destination : REFERENCE TO I_InterfaceDatatype;
END_VAR
Destination := THIS^;
TryResolveAsInterfaceDatatype := TRUE;
END_METHOD

PROPERTY PUBLIC TypeName : T_MAXSTRING
GET
TypeName := 'INTERFACE';
END_GET
END_PROPERTY

END_FUNCTION_BLOCK

// mobject-datatypes/_Internal/Datatype/StructuredDatatypeBase
{attribute 'linkalways'} 
{attribute 'no_explicit_call' := 'This FB is a CLASS and must be accessed using methods or properties'}
{attribute 'enable_dynamic_creation'}
FUNCTION_BLOCK ABSTRACT StructuredDatatypeBase EXTENDS UserDefinedDatatypeBase IMPLEMENTS I_StructuredDatatype
VAR
	membersHost : StructureMemberHost;
END_VAR

METHOD PROTECTED AddMember
VAR_INPUT
	MemberName : T_MAXSTRING;
	Member : I_Datatype;
END_VAR
membersHost.AddMember(MemberName, Member);
END_METHOD

METHOD PROTECTED OnSerializeTypeWith
VAR_INPUT
	Serializer : I_Serializer;
END_VAR
SUPER^.OnSerializeTypeWith(Serializer);
membersHost.SerializeTypeWith(Serializer);
END_METHOD

METHOD PUBLIC Accept
VAR_INPUT
	Visitor : I_DatatypeVisitor;
END_VAR
Visitor.VisitDatatype(THIS^);
membersHost.Accept(Visitor);
END_METHOD

PROPERTY PUBLIC Members : I_StructureMembers
GET
Members := membersHost;
END_GET
END_PROPERTY

METHOD PUBLIC SerializeWith
VAR_INPUT
	Serializer : I_Serializer;
END_VAR
Serializer.StartObject();
membersHost.SerializeWith(Serializer);
Serializer.EndObject();
END_METHOD

METHOD TryDeserializeFrom : BOOL
VAR_INPUT
	Deserializer : I_Deserializer;
	Feedback : I_DeserializerFeedback;
END_VAR
TryDeserializeFrom := membersHost.TryDeserializeFrom(Deserializer, Feedback);
END_METHOD

METHOD PUBLIC TryResolveAsStructuredDatatype : BOOL
VAR_INPUT
	Destination : REFERENCE TO I_StructuredDatatype;
END_VAR
Destination := THIS^;
TryResolveAsStructuredDatatype := TRUE;
END_METHOD

PROPERTY PUBLIC TypeName : T_MAXSTRING
GET
TypeName := 'STRUCT';
END_GET
END_PROPERTY

END_FUNCTION_BLOCK

// mobject-datatypes/_Internal/StructureMembers/Host/StructureMemberHost
{attribute 'linkalways'} 
{attribute 'no_explicit_call' := 'This FB is a CLASS and must be accessed using methods or properties'}
{attribute 'enable_dynamic_creation'}
FUNCTION_BLOCK StructureMemberHost IMPLEMENTS I_Serializable, I_StructureMembers
VAR
	members : OrderedDictionary;
END_VAR

METHOD PUBLIC Accept
VAR_INPUT
	Visitor : I_DatatypeVisitor;
END_VAR
VAR
	enumerator : I_ForwardEnumerator;
	member : I_Datatype;
END_VAR
enumerator := members.GetEnumerator();

WHILE (enumerator.MoveNext()) DO
	
	IF enumerator.TryGet(member) THEN
		member.Accept(Visitor);
	END_IF

END_WHILE

enumerator.Dispose();
END_METHOD

METHOD PUBLIC AddMember
VAR_INPUT
	MemberName : T_MAXSTRING;
	Member : I_Datatype;
END_VAR
members.AddOrUpdate(MemberName, Member);
END_METHOD

METHOD PUBLIC GetMemberEnumerator : I_KeyValueForwardEnumerator
VAR_INPUT
END_VAR
GetMemberEnumerator := members.GetKeyValueEnumerator();
END_METHOD

METHOD PUBLIC SerializeTypeWith
VAR_INPUT
	Serializer : I_Serializer;
END_VAR
VAR
	enumerator : I_KeyValueForwardEnumerator;
	member : I_Datatype;
END_VAR
IF members.Count = 0 THEN
	RETURN;
END_IF

Serializer.AddKey('members');
Serializer.StartObject();

enumerator := members.GetKeyValueEnumerator();

WHILE enumerator.MoveNext() DO
	IF enumerator.TryGet(member) THEN
		Serializer.AddKey(enumerator.Key);
		member.SerializeTypeWith(Serializer);
	END_IF
END_WHILE

enumerator.Dispose();

Serializer.EndObject();
END_METHOD

METHOD PUBLIC SerializeWith
VAR_INPUT
	Serializer : I_Serializer;
END_VAR
VAR
	enumerator : I_KeyValueForwardEnumerator;
	member : I_Datatype;
END_VAR
enumerator := members.GetKeyValueEnumerator();

WHILE enumerator.MoveNext() DO
	IF enumerator.TryGet(member) THEN
		Serializer.AddKey(enumerator.Key);
		member.SerializeWith(Serializer);
	END_IF
END_WHILE

enumerator.Dispose();
END_METHOD

METHOD PUBLIC TryDeserializeFrom : BOOL
VAR_INPUT
	Deserializer : I_Deserializer;
	Feedback : I_DeserializerFeedback;
END_VAR
VAR
	membersEnumerator : I_DeserializerObjectForwardEnumerator;
	member : I_Datatype;
END_VAR
membersEnumerator := Deserializer.GetObjectEnumerator();

WHILE membersEnumerator.MoveNext() DO
	
	IF NOT TryGetMemberByName(membersEnumerator.Key, member) THEN
		CONTINUE;
	END_IF
	
	IF NOT member.TryDeserializeFrom(membersEnumerator.Current, Feedback) THEN
		RETURN;
	END_IF

END_WHILE

membersEnumerator.Dispose();
TryDeserializeFrom := TRUE;
END_METHOD

METHOD PUBLIC TryGetMemberByName : BOOL
VAR_INPUT
	Name : T_MAXSTRING;
	Destination : REFERENCE TO I_Datatype;
END_VAR
VAR
	member : I_Datatype;
END_VAR
IF NOT members.TryGetValue(Name, member) THEN
	RETURN;
END_IF

Destination := member;
TryGetMemberByName := TRUE;
END_METHOD

END_FUNCTION_BLOCK

// mobject-datatypes/_Internal/Events/AliasDatatypeAddedEvent
{attribute 'linkalways'} 
{attribute 'no_explicit_call' := 'This FB is a CLASS and must be accessed using methods or properties'}
{attribute 'enable_dynamic_creation'}
FUNCTION_BLOCK AliasDatatypeAddedEvent EXTENDS Disposable IMPLEMENTS I_AliasDatatypeAddedEvent
VAR
	_target : I_AliasDatatype;
END_VAR

METHOD FB_init : BOOL
VAR_INPUT
	bInitRetains : BOOL; // if TRUE, the retain variables are initialized (warm start / cold start)
	bInCopyCode : BOOL;  // if TRUE, the instance afterwards gets moved into the copy code (online change)
	Target : I_AliasDatatype;
END_VAR
This^._target := Target;
END_METHOD

PROPERTY PUBLIC Target : I_AliasDatatype
GET
Target := _target;
END_GET
END_PROPERTY

END_FUNCTION_BLOCK

// mobject-datatypes/Datatypes/Events/I_AliasDatatypeAddedEvent
INTERFACE I_AliasDatatypeAddedEvent EXTENDS I_Event

PROPERTY PUBLIC Target : I_AliasDatatype
GET
END_GET
END_PROPERTY

END_INTERFACE

// mobject-datatypes/_Internal/Events/ArrayDatatypeAddedEvent
{attribute 'linkalways'} 
{attribute 'no_explicit_call' := 'This FB is a CLASS and must be accessed using methods or properties'}
{attribute 'enable_dynamic_creation'}
FUNCTION_BLOCK ArrayDatatypeAddedEvent EXTENDS Disposable IMPLEMENTS I_ArrayDatatypeAddedEvent
VAR
	_target : I_ArrayDatatype;
END_VAR

METHOD FB_init : BOOL
VAR_INPUT
	bInitRetains : BOOL; // if TRUE, the retain variables are initialized (warm start / cold start)
	bInCopyCode : BOOL;  // if TRUE, the instance afterwards gets moved into the copy code (online change)
	Target : I_ArrayDatatype;
END_VAR
This^._target := Target;
END_METHOD

PROPERTY PUBLIC Target : I_ArrayDatatype
GET
Target := _target;
END_GET
END_PROPERTY

END_FUNCTION_BLOCK

// mobject-datatypes/Datatypes/Events/I_ArrayDatatypeAddedEvent
INTERFACE I_ArrayDatatypeAddedEvent EXTENDS I_Event

PROPERTY PUBLIC Target : I_ArrayDatatype
GET
END_GET
END_PROPERTY

END_INTERFACE

// mobject-datatypes/_Internal/Events/DatatypeAddedEvent
{attribute 'linkalways'} 
{attribute 'no_explicit_call' := 'This FB is a CLASS and must be accessed using methods or properties'}
{attribute 'enable_dynamic_creation'}
FUNCTION_BLOCK DatatypeAddedEvent EXTENDS Disposable IMPLEMENTS I_DatatypeAddedEvent
VAR
	_target : I_Datatype;
END_VAR

METHOD FB_init : BOOL
VAR_INPUT
	bInitRetains : BOOL; // if TRUE, the retain variables are initialized (warm start / cold start)
	bInCopyCode : BOOL;  // if TRUE, the instance afterwards gets moved into the copy code (online change)
	Target : I_Datatype;
END_VAR
This^._target := Target;
END_METHOD

PROPERTY PUBLIC Target : I_Datatype
GET
Target := _target;
END_GET
END_PROPERTY

END_FUNCTION_BLOCK

// mobject-datatypes/Datatypes/Events/I_DatatypeAddedEvent
INTERFACE I_DatatypeAddedEvent EXTENDS I_Event

PROPERTY PUBLIC Target : I_Datatype
GET
END_GET
END_PROPERTY

END_INTERFACE

// mobject-datatypes/_Internal/Events/EnumDatatypeAddedEvent
{attribute 'linkalways'} 
{attribute 'no_explicit_call' := 'This FB is a CLASS and must be accessed using methods or properties'}
{attribute 'enable_dynamic_creation'}
FUNCTION_BLOCK EnumDatatypeAddedEvent EXTENDS Disposable IMPLEMENTS I_EnumDatatypeAddedEvent
VAR
	_target : I_EnumDatatype;
END_VAR

METHOD FB_init : BOOL
VAR_INPUT
	bInitRetains : BOOL; // if TRUE, the retain variables are initialized (warm start / cold start)
	bInCopyCode : BOOL;  // if TRUE, the instance afterwards gets moved into the copy code (online change)
	Target : I_EnumDatatype;
END_VAR
This^._target := Target;
END_METHOD

PROPERTY PUBLIC Target : I_EnumDatatype
GET
Target := _target;
END_GET
END_PROPERTY

END_FUNCTION_BLOCK

// mobject-datatypes/Datatypes/Events/I_EnumDatatypeAddedEvent
INTERFACE I_EnumDatatypeAddedEvent EXTENDS I_Event

PROPERTY PUBLIC Target : I_EnumDatatype
GET
END_GET
END_PROPERTY

END_INTERFACE

// mobject-datatypes/_Internal/Events/InterfaceDatatypeAddedEvent
{attribute 'linkalways'} 
{attribute 'no_explicit_call' := 'This FB is a CLASS and must be accessed using methods or properties'}
{attribute 'enable_dynamic_creation'}
FUNCTION_BLOCK InterfaceDatatypeAddedEvent EXTENDS Disposable IMPLEMENTS I_InterfaceDatatypeAddedEvent
VAR
	_target : I_InterfaceDatatype;
END_VAR

METHOD FB_init : BOOL
VAR_INPUT
	bInitRetains : BOOL; // if TRUE, the retain variables are initialized (warm start / cold start)
	bInCopyCode : BOOL;  // if TRUE, the instance afterwards gets moved into the copy code (online change)
	Target : I_InterfaceDatatype;
END_VAR
This^._target := Target;
END_METHOD

PROPERTY PUBLIC Target : I_InterfaceDatatype
GET
Target := _target;
END_GET
END_PROPERTY

END_FUNCTION_BLOCK

// mobject-datatypes/Datatypes/Events/I_InterfaceDatatypeAddedEvent
INTERFACE I_InterfaceDatatypeAddedEvent EXTENDS I_Event

PROPERTY PUBLIC Target : I_InterfaceDatatype
GET
END_GET
END_PROPERTY

END_INTERFACE

// mobject-datatypes/_Internal/Events/StructuredDatatypeAddedEvent
{attribute 'linkalways'} 
{attribute 'no_explicit_call' := 'This FB is a CLASS and must be accessed using methods or properties'}
{attribute 'enable_dynamic_creation'}
FUNCTION_BLOCK StructuredDatatypeAddedEvent EXTENDS Disposable IMPLEMENTS I_StructuredDatatypeAddedEvent
VAR
	_target : I_StructuredDatatype;
END_VAR

METHOD FB_init : BOOL
VAR_INPUT
	bInitRetains : BOOL; // if TRUE, the retain variables are initialized (warm start / cold start)
	bInCopyCode : BOOL;  // if TRUE, the instance afterwards gets moved into the copy code (online change)
	Target : I_StructuredDatatype;
END_VAR
This^._target := Target;
END_METHOD

PROPERTY PUBLIC Target : I_StructuredDatatype
GET
Target := _target;
END_GET
END_PROPERTY

END_FUNCTION_BLOCK

// mobject-datatypes/Datatypes/Events/I_StructuredDatatypeAddedEvent
INTERFACE I_StructuredDatatypeAddedEvent EXTENDS I_Event

PROPERTY PUBLIC Target : I_StructuredDatatype
GET
END_GET
END_PROPERTY

END_INTERFACE

// mobject-datatypes/DatatypeOperations/Collection/DatatypeOperations
{attribute 'linkalways'} 
{attribute 'no_explicit_call' := 'This FB is a CLASS and must be accessed using methods or properties'}
{attribute 'enable_dynamic_creation'}
FUNCTION_BLOCK DatatypeOperations
VAR
	operations : Stack;
END_VAR

METHOD FB_exit : BOOL
VAR_INPUT
	bInCopyCode : BOOL; // if TRUE, the exit method is called for exiting an instance that is copied afterwards (online change).
END_VAR
IF bInCopyCode THEN
	RETURN;
END_IF

operations.Clear();
END_METHOD

METHOD PRIVATE CreateMemoryCopyOperation : I_DatatypeOperation
VAR_INPUT
	OperationSource : I_Datatype;
	OperationDestination : I_Datatype;
END_VAR
VAR
	pOperation : POINTER TO MemCopyOperation;
END_VAR
pOperation := __NEW(MemCopyOperation(Source := OperationSource, Destination := OperationDestination));
CreateMemoryCopyOperation := pOperation^;
END_METHOD

METHOD PRIVATE CreateSafeMemoryCopyOperation : I_DatatypeOperation
VAR_INPUT
	OperationSource : I_Datatype;
	OperationDestination : I_Datatype;
END_VAR
VAR
	pOperation : POINTER TO SafeMemCopyOperation;
END_VAR
pOperation := __NEW(SafeMemCopyOperation(Source := OperationSource, Destination := OperationDestination));
CreateSafeMemoryCopyOperation := pOperation^;
END_METHOD

METHOD PRIVATE CreateWriteBitToBoolOperation : I_DatatypeOperation
VAR_INPUT
	OperationSource : I_BitDatatype;
	OperationDestination : REFERENCE TO _BOOL;
END_VAR
VAR
	pOperation : POINTER TO WriteBitToBoolOperation;
END_VAR
pOperation := __NEW(WriteBitToBoolOperation(Source := OperationSource, Destination := OperationDestination));
CreateWriteBitToBoolOperation := pOperation^;
END_METHOD

METHOD PRIVATE CreateWriteBoolToBitOperation : I_DatatypeOperation
VAR_INPUT
	OperationSource : REFERENCE TO _BOOL;
	OperationDestination : I_BitDatatype;
END_VAR
VAR
	pOperation : POINTER TO WriteBoolToBitOperation;
END_VAR
pOperation := __NEW(WriteBoolToBitOperation(Source := OperationSource, Destination := OperationDestination));
CreateWriteBoolToBitOperation := pOperation^;
END_METHOD

METHOD PUBLIC AddMemoryCopyOperation
VAR_INPUT
	Source : I_Datatype;
	Destination : I_Datatype;
END_VAR
VAR
	operation : I_DatatypeOperation;
END_VAR
operation := CreateMemoryCopyOperation(Source,Destination);
operations.Push(operation);
END_METHOD

METHOD PUBLIC AddSafeMemoryCopyOperation
VAR_INPUT
	Source : I_Datatype;
	Destination : I_Datatype;
END_VAR
VAR
	operation : I_DatatypeOperation;
END_VAR
operation := CreateSafeMemoryCopyOperation(Source,Destination);
operations.Push(operation);
END_METHOD

METHOD PUBLIC AddWriteBitToBoolOperation
VAR_INPUT
	Source : I_BitDatatype;
	Destination : Reference to _BOOL;
END_VAR
VAR
	operation : I_DatatypeOperation;
END_VAR
operation := CreateWriteBitToBoolOperation(Source,Destination);
operations.Push(operation);
END_METHOD

METHOD PUBLIC AddWriteBoolToBitOperation
VAR_INPUT
	Source : REFERENCE TO _BOOL;
	Destination : I_BitDatatype;
END_VAR
VAR
	operation : I_DatatypeOperation;
END_VAR
operation := CreateWriteBoolToBitOperation(Source,Destination);
operations.Push(operation);
END_METHOD

METHOD PUBLIC Clear
VAR
	operation : I_DatatypeOperation;
END_VAR
WHILE operations.TryPop(operation) DO
	operation.Dispose();
END_WHILE
END_METHOD

METHOD PUBLIC Execute
VAR
	enumerator : I_ForwardEnumerator;
	operation : I_DatatypeOperation;
END_VAR
enumerator := operations.GetEnumerator();

WHILE enumerator.MoveNext() DO
	IF enumerator.TryGet(operation) THEN
		operation.Execute();
	END_IF
END_WHILE

enumerator.Dispose();
END_METHOD

END_FUNCTION_BLOCK

// mobject-datatypes/DatatypeOperations/MemCopyOperation
{attribute 'linkalways'} 
{attribute 'no_explicit_call' := 'This FB is a CLASS and must be accessed using methods or properties'}
{attribute 'enable_dynamic_creation'}
FUNCTION_BLOCK MemCopyOperation EXTENDS Disposable IMPLEMENTS I_DatatypeOperation
VAR
	source : I_Datatype;
	destination : I_Datatype;
END_VAR

METHOD FB_init : BOOL
VAR_INPUT
	bInitRetains : BOOL; // if TRUE, the retain variables are initialized (warm start / cold start)
	bInCopyCode : BOOL;  // if TRUE, the instance afterwards gets moved into the copy code (online change)
	Source : I_Datatype;
	Destination : I_Datatype;
END_VAR
THIS^.source := Source;
This^.destination := Destination;
END_METHOD

METHOD Execute
VAR
END_VAR
memcpy(destination.Address, source.Address, source.Size);
END_METHOD

END_FUNCTION_BLOCK

// mobject-datatypes/DatatypeOperations/Interface/I_DatatypeOperation
INTERFACE I_DatatypeOperation EXTENDS I_Disposable

METHOD Execute
VAR
END_VAR
END_METHOD

END_INTERFACE

// mobject-datatypes/DatatypeOperations/SafeMemCopyOperation
{attribute 'linkalways'} 
{attribute 'no_explicit_call' := 'This FB is a CLASS and must be accessed using methods or properties'}
{attribute 'enable_dynamic_creation'}
FUNCTION_BLOCK SafeMemCopyOperation EXTENDS Disposable IMPLEMENTS I_DatatypeOperation
VAR
	source : I_Datatype;
	destination : I_Datatype;
END_VAR

METHOD FB_init : BOOL
VAR_INPUT
	bInitRetains : BOOL; // if TRUE, the retain variables are initialized (warm start / cold start)
	bInCopyCode : BOOL;  // if TRUE, the instance afterwards gets moved into the copy code (online change)
	Source : I_Datatype;
	Destination : I_Datatype;
END_VAR
THIS^.source := Source;
This^.destination := Destination;
END_METHOD

METHOD Execute
VAR
END_VAR
destination.TryCopyFrom(source);
END_METHOD

END_FUNCTION_BLOCK

// mobject-datatypes/DatatypeOperations/WriteBitToBoolOperation
{attribute 'linkalways'} 
{attribute 'no_explicit_call' := 'This FB is a CLASS and must be accessed using methods or properties'}
{attribute 'enable_dynamic_creation'}
FUNCTION_BLOCK WriteBitToBoolOperation EXTENDS Disposable IMPLEMENTS I_DatatypeOperation
VAR
	source : I_BitDatatype;
	destination : REFERENCE TO _BOOL;
END_VAR

METHOD FB_init : BOOL
VAR_INPUT
	bInitRetains : BOOL; // if TRUE, the retain variables are initialized (warm start / cold start)
	bInCopyCode : BOOL;  // if TRUE, the instance afterwards gets moved into the copy code (online change)
	Source : I_BitDatatype;
	Destination : REFERENCE TO _BOOL;
END_VAR
THIS^.source := Source;
THIS^.destination REF= Destination;
END_METHOD

METHOD Execute
VAR
END_VAR
destination.Value := source.Value;
END_METHOD

END_FUNCTION_BLOCK

// mobject-datatypes/DatatypeOperations/WriteBoolToBitOperation
{attribute 'linkalways'} 
{attribute 'no_explicit_call' := 'This FB is a CLASS and must be accessed using methods or properties'}
{attribute 'enable_dynamic_creation'}
FUNCTION_BLOCK WriteBoolToBitOperation EXTENDS Disposable IMPLEMENTS I_DatatypeOperation
VAR
	source : REFERENCE TO _BOOL;
	destination : I_BitDatatype;
END_VAR

METHOD FB_init : BOOL
VAR_INPUT
	bInitRetains : BOOL; // if TRUE, the retain variables are initialized (warm start / cold start)
	bInCopyCode : BOOL;  // if TRUE, the instance afterwards gets moved into the copy code (online change)
	Source : REFERENCE TO _BOOL;
	Destination : I_BitDatatype;
END_VAR
THIS^.source REF= Source;
THIS^.destination := Destination;
END_METHOD

METHOD Execute
VAR
END_VAR
destination.Value := source.Value;
END_METHOD

END_FUNCTION_BLOCK

// mobject-datatypes/Datatypes/Base/Datatypes
{attribute 'linkalways'} 
{attribute 'no_explicit_call' := 'This FB is a CLASS and must be accessed using methods or properties'}
{attribute 'enable_dynamic_creation'}
FUNCTION_BLOCK Datatypes IMPLEMENTS I_Datatypes
VAR
	eventEmitter : EventEmitter;
	primitives : Dictionary;
	structures : Dictionary;
	arrays : Dictionary;
	alias : Dictionary;
	enums : Dictionary;
	interfaces : Dictionary;
END_VAR

METHOD PRIVATE AcceptAlias
VAR_INPUT
	Visitor : I_DatatypeVisitor;
END_VAR
VAR
	enumerator : I_ForwardEnumerator;
	datatype : I_AliasDatatype;
END_VAR
enumerator := alias.GetEnumerator();

WHILE enumerator.MoveNext() DO
	IF enumerator.TryGet(datatype) THEN
		datatype.Accept(Visitor);
	END_IF
END_WHILE

enumerator.Dispose();
END_METHOD

METHOD PRIVATE AcceptArrays
VAR_INPUT
	Visitor : I_DatatypeVisitor;
END_VAR
VAR
	enumerator : I_ForwardEnumerator;
	datatype : I_ArrayDatatype;
END_VAR
enumerator := arrays.GetEnumerator();

WHILE enumerator.MoveNext() DO	
	IF enumerator.TryGet(datatype) THEN
		datatype.Accept(Visitor);
	END_IF
END_WHILE

enumerator.Dispose();
END_METHOD

METHOD PRIVATE AcceptEnum
VAR_INPUT
	Visitor : I_DatatypeVisitor;
END_VAR
VAR
	enumerator : I_ForwardEnumerator;
	datatype : I_EnumDatatype;
END_VAR
enumerator := enums.GetEnumerator();

WHILE enumerator.MoveNext() DO
	IF enumerator.TryGet(datatype) THEN
		datatype.Accept(Visitor);
	END_IF
END_WHILE

enumerator.Dispose();
END_METHOD

METHOD PRIVATE AcceptInterface
VAR_INPUT
	Visitor : I_DatatypeVisitor;
END_VAR
VAR
	enumerator : I_ForwardEnumerator;
	datatype : I_InterfaceDatatype;
END_VAR
enumerator := structures.GetEnumerator();

WHILE enumerator.MoveNext() DO	
	IF enumerator.TryGet(datatype) THEN
		datatype.Accept(Visitor);
	END_IF
END_WHILE

enumerator.Dispose();
END_METHOD

METHOD PRIVATE AcceptPrimative
VAR_INPUT
	Visitor : I_DatatypeVisitor;
END_VAR
VAR
	enumerator : I_ForwardEnumerator;
	datatype : I_Datatype;
END_VAR
enumerator := primitives.GetEnumerator();

WHILE enumerator.MoveNext() DO
	IF enumerator.TryGet(datatype) THEN
		datatype.Accept(Visitor);
	END_IF
END_WHILE

enumerator.Dispose();
END_METHOD

METHOD PRIVATE AcceptStructures
VAR_INPUT
	Visitor : I_DatatypeVisitor;
END_VAR
VAR
	enumerator : I_ForwardEnumerator;
	datatype : I_StructuredDatatype;
END_VAR
enumerator := structures.GetEnumerator();

WHILE enumerator.MoveNext() DO	
	IF enumerator.TryGet(datatype) THEN
		datatype.Accept(Visitor);
	END_IF
END_WHILE

enumerator.Dispose();
END_METHOD

METHOD PRIVATE SerializeAliasTypeWith
VAR_INPUT
	Serializer : I_Serializer;
END_VAR
VAR
	enumerator : I_ForwardEnumerator;
	datatype : I_AliasDatatype;
END_VAR
enumerator := alias.GetEnumerator();

WHILE enumerator.MoveNext() DO
	IF enumerator.TryGet(datatype) THEN
		datatype.SerializeTypeWith(Serializer);
	END_IF
END_WHILE

enumerator.Dispose();
END_METHOD

METHOD PRIVATE SerializeArrayTypeWith
VAR_INPUT
	Serializer : I_Serializer;
END_VAR
VAR
	enumerator : I_ForwardEnumerator;
	datatype : I_ArrayDatatype;
END_VAR
enumerator := arrays.GetEnumerator();

WHILE enumerator.MoveNext() DO
	IF enumerator.TryGet(datatype) THEN
		datatype.SerializeTypeWith(Serializer);
	END_IF
END_WHILE

enumerator.Dispose();
END_METHOD

METHOD PRIVATE SerializeEnumsTypeWith
VAR_INPUT
	Serializer : I_Serializer;
END_VAR
VAR
	enumerator : I_ForwardEnumerator;
	datatype : I_EnumDatatype;
END_VAR
enumerator := enums.GetEnumerator();

WHILE enumerator.MoveNext() DO
	IF enumerator.TryGet(datatype) THEN
		datatype.SerializeTypeWith(Serializer);
	END_IF
END_WHILE

enumerator.Dispose();
END_METHOD

METHOD PRIVATE SerializeInterfaceTypeWith
VAR_INPUT
	Serializer : I_Serializer;
END_VAR
VAR
	enumerator : I_ForwardEnumerator;
	datatype : I_InterfaceDatatype;
END_VAR
enumerator := interfaces.GetEnumerator();

WHILE enumerator.MoveNext() DO
	IF enumerator.TryGet(datatype) THEN
		datatype.SerializeTypeWith(Serializer);
	END_IF
END_WHILE

enumerator.Dispose();
END_METHOD

METHOD PRIVATE SerializePrimitiveTypeWith
VAR_INPUT
	Serializer : I_Serializer;
END_VAR
VAR
	enumerator : I_ForwardEnumerator;
	datatype : I_Datatype;
END_VAR
enumerator := primitives.GetEnumerator();

WHILE enumerator.MoveNext() DO
	IF enumerator.TryGet(datatype) THEN
		datatype.SerializeTypeWith(Serializer);
	END_IF
END_WHILE

enumerator.Dispose();
END_METHOD

METHOD PRIVATE SerializeStructuresTypeWith
VAR_INPUT
	Serializer : I_Serializer;
END_VAR
VAR
	enumerator : I_ForwardEnumerator;
	datatype : I_StructuredDatatype;
END_VAR
enumerator := structures.GetEnumerator();

WHILE enumerator.MoveNext() DO
	IF enumerator.TryGet(datatype) THEN
		datatype.SerializeTypeWith(Serializer);
	END_IF
END_WHILE

enumerator.Dispose();
END_METHOD

METHOD PROTECTED EmitOnAliasDatatypeAddedEvent
VAR_INPUT
	Datatype : I_AliasDatatype;
END_VAR
VAR
	datatypeAddedEvent : AliasDatatypeAddedEvent(Target := Datatype);
END_VAR
eventEmitter.Emit('OnDatatypeAdded', datatypeAddedEvent);
END_METHOD

METHOD PROTECTED EmitOnArrayDatatypeAddedEvent
VAR_INPUT
	Datatype : I_ArrayDatatype;
END_VAR
VAR
	datatypeAddedEvent : ArrayDatatypeAddedEvent(Target := Datatype);
END_VAR
eventEmitter.Emit('OnDatatypeAdded', datatypeAddedEvent);
END_METHOD

METHOD PROTECTED EmitOnDatatypeAddedEvent
VAR_INPUT
	Datatype : I_Datatype;
END_VAR
VAR
	datatypeAddedEvent : DatatypeAddedEvent(Target := Datatype);
END_VAR
eventEmitter.Emit('OnDatatypeAdded', datatypeAddedEvent);
END_METHOD

METHOD PROTECTED EmitOnEnumDatatypeAddedEvent
VAR_INPUT
	Datatype : I_EnumDatatype;
END_VAR
VAR
	datatypeAddedEvent : EnumDatatypeAddedEvent(Target := Datatype);
END_VAR
eventEmitter.Emit('OnDatatypeAdded', datatypeAddedEvent);
END_METHOD

METHOD PROTECTED EmitOnInterfaceDatatypeAddedEvent
VAR_INPUT
	Datatype : I_InterfaceDatatype;
END_VAR
VAR
	datatypeAddedEvent : InterfaceDatatypeAddedEvent(Target := Datatype);
END_VAR
eventEmitter.Emit('OnDatatypeAdded', datatypeAddedEvent);
END_METHOD

METHOD PROTECTED EmitOnStructuredDatatypeAddedEvent
VAR_INPUT
	Datatype : I_StructuredDatatype;
END_VAR
VAR
	datatypeAddedEvent : StructuredDatatypeAddedEvent(Target := Datatype);
END_VAR
eventEmitter.Emit('OnDatatypeAdded', datatypeAddedEvent);
END_METHOD

METHOD PUBLIC Accept
VAR_INPUT
	Visitor : I_DatatypeVisitor;
END_VAR
AcceptPrimative(Visitor);
AcceptStructures(Visitor);
AcceptArrays(Visitor);
AcceptAlias(Visitor);
AcceptEnum(Visitor);
AcceptInterface(Visitor);
END_METHOD

METHOD PUBLIC OffEvent
VAR_INPUT
	EventName : T_MaxString;
	EventHandler : I_EventHandler;
END_VAR
eventEmitter.OffEvent(EventName, EventHandler);
END_METHOD

METHOD PUBLIC OnceEvent
VAR_INPUT
	EventName : T_MaxString;
	EventHandler : I_EventHandler;
END_VAR
eventEmitter.OnceEvent(EventName, EventHandler);
END_METHOD

METHOD PUBLIC OnEvent
VAR_INPUT
	EventName : T_MaxString;
	EventHandler : I_EventHandler;
END_VAR
eventEmitter.OnEvent(EventName, EventHandler);
END_METHOD

METHOD RegisterDatatype
VAR_INPUT
	Datatype : I_Datatype;
END_VAR
VAR
	datatypeAsStructure : I_StructuredDatatype;
	datatypeAsArray : I_ArrayDatatype;
	datatypeAsAlias : I_AliasDatatype;
	datatypeAsEnum : I_EnumDatatype;
	datatypeAsInterface : I_InterfaceDatatype;
END_VAR
IF Datatype.TryResolveAsStructuredDatatype(datatypeAsStructure) THEN
	structures.AddOrUpdate(datatypeAsStructure.Identifier, datatypeAsStructure);
	emitOnStructuredDatatypeAddedEvent(datatypeAsStructure);
	RETURN;
END_IF

IF Datatype.TryResolveAsArrayDatatype(datatypeAsArray) THEN
	arrays.AddOrUpdate(datatypeAsArray.Identifier, datatypeAsArray);
	emitOnArrayDatatypeAddedEvent(datatypeAsArray);
	RETURN;
END_IF

IF Datatype.TryResolveAsAliasDatatype(datatypeAsAlias) THEN
	alias.AddOrUpdate(datatypeAsAlias.Identifier, datatypeAsAlias);
	emitOnAliasDatatypeAddedEvent(datatypeAsAlias);
	RETURN;
END_IF

IF Datatype.TryResolveAsEnumDatatype(datatypeAsEnum) THEN
	enums.AddOrUpdate(datatypeAsEnum.Identifier, datatypeAsEnum);
	emitOnEnumDatatypeAddedEvent(datatypeAsEnum);
	RETURN;
END_IF

IF Datatype.TryResolveAsInterfaceDatatype(datatypeAsInterface) THEN
	interfaces.AddOrUpdate(datatypeAsInterface.Identifier, datatypeAsInterface);
	emitOnInterfaceDatatypeAddedEvent(datatypeAsInterface);
	RETURN;
END_IF

primitives.AddOrUpdate(Datatype.TypeName, Datatype);
emitOnDatatypeAddedEvent(Datatype);
END_METHOD

METHOD PUBLIC SerializeTypeWith
VAR_INPUT
	Serializer : I_Serializer;
END_VAR
Serializer.StartObject();
Serializer.AddKey('datatypes');
Serializer.StartArray();
SerializePrimitiveTypeWith(Serializer);
SerializeStructuresTypeWith(Serializer);
SerializeArrayTypeWith(Serializer);
SerializeAliasTypeWith(Serializer);
SerializeEnumsTypeWith(Serializer);
SerializeInterfaceTypeWith(Serializer);
Serializer.EndArray();
Serializer.EndObject();
END_METHOD

METHOD PUBLIC TryGetAliasByIdentifier : BOOL
VAR_INPUT
	Identifier : T_MAXSTRING;
	Destination : REFERENCE TO I_AliasDatatype;
END_VAR
TryGetAliasByIdentifier := alias.TryGetValue(Identifier, Destination);
END_METHOD

METHOD PUBLIC TryGetArrayByIdentifier : BOOL
VAR_INPUT
	Identifier : T_MAXSTRING;
	Destination : REFERENCE TO I_ArrayDatatype;
END_VAR
TryGetArrayByIdentifier := arrays.TryGetValue(Identifier, Destination);
END_METHOD

METHOD PUBLIC TryGetEnumByIdentifier : BOOL
VAR_INPUT
	Identifier : T_MAXSTRING;
	Destination : REFERENCE TO I_EnumDatatype;
END_VAR
TryGetEnumByIdentifier := enums.TryGetValue(Identifier, Destination);
END_METHOD

METHOD PUBLIC TryGetInterfaceByIdentifier : BOOL
VAR_INPUT
	Identifier : T_MAXSTRING;
	Destination : REFERENCE TO I_InterfaceDatatype;
END_VAR
TryGetInterfaceByIdentifier := interfaces.TryGetValue(Identifier, Destination);
END_METHOD

METHOD PUBLIC TryGetPrimitiveByTypeName : BOOL
VAR_INPUT
	TypeName : T_MAXSTRING;
	Destination : REFERENCE TO I_AliasDatatype;
END_VAR
TryGetPrimitiveByTypeName := primitives.TryGetValue(TypeName, Destination);
END_METHOD

METHOD PUBLIC TryGetStructureByIdentifier : BOOL
VAR_INPUT
	Identifier : T_MAXSTRING;
	Destination : REFERENCE TO I_StructuredDatatype;
END_VAR
TryGetStructureByIdentifier := structures.TryGetValue(Identifier, Destination);
END_METHOD

END_FUNCTION_BLOCK

// mobject-datatypes/Datatypes/Interface/I_Datatypes
INTERFACE I_Datatypes EXTENDS I_EventEmitter

METHOD PUBLIC Accept
VAR_INPUT
	Visitor : I_DatatypeVisitor;
END_VAR
END_METHOD

METHOD RegisterDatatype
VAR_INPUT
	Datatype : I_Datatype;
END_VAR
END_METHOD

METHOD PUBLIC SerializeTypeWith
VAR_INPUT
	Serializer : I_Serializer;
END_VAR
END_METHOD

METHOD PUBLIC TryGetAliasByIdentifier : BOOL
VAR_INPUT
	Identifier : T_MAXSTRING;
	Destination : REFERENCE TO I_AliasDatatype;
END_VAR
END_METHOD

METHOD PUBLIC TryGetArrayByIdentifier : BOOL
VAR_INPUT
	Identifier : T_MAXSTRING;
	Destination : REFERENCE TO I_ArrayDatatype;
END_VAR
END_METHOD

METHOD PUBLIC TryGetEnumByIdentifier : BOOL
VAR_INPUT
	Identifier : T_MAXSTRING;
	Destination : REFERENCE TO I_EnumDatatype;
END_VAR
END_METHOD

METHOD PUBLIC TryGetInterfaceByIdentifier : BOOL
VAR_INPUT
	Identifier : T_MAXSTRING;
	Destination : REFERENCE TO I_InterfaceDatatype;
END_VAR
END_METHOD

METHOD PUBLIC TryGetPrimitiveByTypeName : BOOL
VAR_INPUT
	TypeName : T_MAXSTRING;
	Destination : REFERENCE TO I_AliasDatatype;
END_VAR
END_METHOD

METHOD PUBLIC TryGetStructureByIdentifier : BOOL
VAR_INPUT
	Identifier : T_MAXSTRING;
	Destination : REFERENCE TO I_StructuredDatatype;
END_VAR
END_METHOD

END_INTERFACE

// mobject-datatypes/Examples/1DimArray/_Array0to10OfBool
{attribute 'linkalways'} 
{attribute 'no_explicit_call' := 'This FB is a CLASS and must be accessed using methods or properties'}
{attribute 'enable_dynamic_creation'}
FUNCTION_BLOCK _Array0to10OfBool EXTENDS ArrayDatatypeBase
VAR CONSTANT
	lBound : DINT := 0;
	uBound : DINT := 10;
END_VAR
VAR
	localData : ARRAY [lBound..uBound] OF BOOL;
	activeData : REFERENCE TO ARRAY [lBound..uBound] OF BOOL REF= localData;
	elements : ARRAY [lBound..uBound] OF _BOOL(FALSE);
	baseType : _BOOL(FALSE);
END_VAR

METHOD FB_init : BOOL
VAR_INPUT
	bInitRetains : BOOL; // if TRUE, the retain variables are initialized (warm start / cold start)
	bInCopyCode : BOOL;  // if TRUE, the instance afterwards gets moved into the copy code (online change)
END_VAR
SetElementReference();
END_METHOD

METHOD PROTECTED OnSerializeArrayValues
VAR_INPUT
	Serializer : I_Serializer;
END_VAR
VAR
	i : DINT;
END_VAR
FOR i := lBound TO uBound DO
	elements[i].SerializeWith(Serializer);
END_FOR
END_METHOD

METHOD PROTECTED SetElementReference
VAR_INPUT
END_VAR
VAR
	i : DINT;
END_VAR
FOR i := lBound TO uBound DO
	elements[i].MakeReferenceTo(activeData[i]);
END_FOR
END_METHOD

METHOD PROTECTED TryDeserializeArrayValues : BOOL
VAR_INPUT
	Deserializer : I_Deserializer;
	Feedback : I_DeserializerFeedback;
END_VAR
VAR
	enumerator : I_DeserializerArrayForwardEnumerator;
	i : DINT;
END_VAR
enumerator := Deserializer.GetArrayEnumerator();
i := lBound;

WHILE enumerator.MoveNext() AND i <= uBound DO
	
	IF NOT elements[i].TryDeserializeFrom(enumerator.Current, Feedback) THEN
		EXIT;
	END_IF
	i := i + 1;

END_WHILE
enumerator.Dispose();
END_METHOD

PROPERTY PUBLIC Address : PVOID
GET
Address := ADR(activeData);
END_GET
END_PROPERTY

PROPERTY PUBLIC BaseDatatype : I_Datatype
GET
BaseDatatype := baseType;
END_GET
END_PROPERTY

METHOD PUBLIC ClearReference
VAR_INPUT
END_VAR
activeData REF= localData;
SetElementReference();
END_METHOD

METHOD PUBLIC GetElementAsDatatypeByIndex : I_Datatype
VAR_INPUT
	Index : DINT;
END_VAR
GetElementAsDatatypeByIndex := elements[Index];
END_METHOD

PROPERTY PUBLIC LowerBound : DINT
GET
LowerBound := lBound;
END_GET
END_PROPERTY

PROPERTY PUBLIC Size : UDINT
GET
Size := SIZEOF(activeData);
END_GET
END_PROPERTY

PROPERTY PUBLIC UpperBound : DINT
GET
UpperBound := ubound;
END_GET
END_PROPERTY

METHOD PUBLIC Clone : I_Datatype
VAR
    pClone : POINTER TO _Array0to10OfBool;
END_VAR
pClone := __NEW(_Array0to10OfBool());
pClone^.Value := Value;
Clone := pClone^;
END_METHOD

METHOD PUBLIC GetElementByIndex : REFERENCE TO _BOOL;
VAR_INPUT
	Index : DINT;
END_VAR
GetElementByIndex REF= elements[Index];
END_METHOD

METHOD PUBLIC MakeReferenceTo
VAR_INPUT
	ReferenceTarget : REFERENCE TO ARRAY [lBound..uBound] OF BOOL;
END_VAR
activeData REF= ReferenceTarget;
SetElementReference();
END_METHOD

METHOD TryMakeReferenceTo : BOOL
VAR_INPUT
	Target : I_Datatype;
END_VAR
VAR
	targetAsArray : I_ArrayDatatype;
	pTargetData : POINTER TO ARRAY [lBound..uBound] OF BOOL;
END_VAR
IF NOT Target.TryResolveAsArrayDatatype(targetAsArray) THEN
	RETURN;
END_IF

IF NOT (targetAsArray.Identifier = Identifier) THEN
	RETURN;
END_IF

pTargetData := Target.Address;
activeData REF= pTargetData^;
SetElementReference();
TryMakeReferenceTo := TRUE;
END_METHOD

PROPERTY PUBLIC Value : REFERENCE TO ARRAY [lBound..uBound] OF BOOL;
GET
Value ref= activeData;
END_GET
END_PROPERTY

END_FUNCTION_BLOCK

// mobject-datatypes/Functions/GetByteOffset
{attribute 'linkalways'} 
FUNCTION GetByteOffset : PVOID
VAR_INPUT
	Structure : ANY;
	Member : ANY_BIT; 
END_VAR

GetByteOffset := Member.pValue - Structure.pValue;

END_FUNCTION

// mobject-datatypes/Primitive/_BIT
{attribute 'linkalways'} 
{attribute 'no_explicit_call' := 'This FB is a CLASS and must be accessed using methods or properties'}
{attribute 'enable_dynamic_creation'}
FUNCTION_BLOCK _BIT EXTENDS DatatypeBase implements I_BitDatatype
VAR
	initialised : BOOL;
	activeParent : I_StructuredDatatype;
	activeByteOffset : PVOID;
	activeBitOffset : DWORD;
END_VAR

METHOD PRIVATE GetBitValue : BOOL
VAR
	pByte : POINTER TO BYTE := Address;
END_VAR
IF NOT initialised THEN
	RETURN;
END_IF

CASE activeBitOffset OF
	0: GetBitValue := pByte^.0;
	1: GetBitValue := pByte^.1;
	2: GetBitValue := pByte^.2;
	3: GetBitValue := pByte^.3;
	4: GetBitValue := pByte^.4;
	5: GetBitValue := pByte^.5;
	6: GetBitValue := pByte^.6;
	7: GetBitValue := pByte^.7;
END_CASE;
END_METHOD

METHOD PRIVATE SetBitValue : BOOL
VAR_INPUT
	Value : BOOL;
END_VAR
VAR
	pByte : POINTER TO BYTE := Address;
END_VAR
IF NOT initialised THEN
	RETURN;
END_IF

CASE activeBitOffset OF
	0: pByte^.0 := Value;
	1: pByte^.1 := Value;
	2: pByte^.2 := Value;
	3: pByte^.3 := Value;
	4: pByte^.4 := Value;
	5: pByte^.5 := Value;
	6: pByte^.6 := Value;
	7: pByte^.7 := Value;
END_CASE;
END_METHOD

PROPERTY PUBLIC Address : PVOID
GET
IF NOT initialised THEN 
	RETURN;
END_IF

Address := activeParent.Address + activeByteOffset;
END_GET
END_PROPERTY

PROPERTY PUBLIC BitOffset : DWORD
GET
IF NOT initialised THEN 
	RETURN;
END_IF

BitOffset := activeBitOffset;
END_GET
END_PROPERTY

PROPERTY PUBLIC ByteOffset : PVOID
GET
IF NOT initialised THEN 
	RETURN;
END_IF

ByteOffset := activeByteOffset;
END_GET
END_PROPERTY

METHOD PUBLIC ClearReference
VAR_INPUT
END_VAR
activeParent := 0;
activeByteOffset := 0;
activeBitOffset := 0;
initialised := FALSE;
END_METHOD

METHOD PUBLIC Clone : I_Datatype
VAR
    pClone : POINTER TO _BIT;
END_VAR
pClone := __NEW(_BIT);

IF initialised THEN
	pClone^.MakeReferenceTo(activeParent, activeByteOffset, activeBitOffset);
END_IF

Clone := pClone^;
END_METHOD

METHOD PUBLIC MakeReferenceTo
VAR_INPUT
	Parent : I_StructuredDatatype;
	ByteOffset : PVOID;
	BitOffset : DWORD;
END_VAR
activeParent := Parent;
activeByteOffset := ByteOffset;
activeBitOffset := BitOffset AND 16#7;
initialised := TRUE;
END_METHOD

PROPERTY PUBLIC Parent : I_StructuredDatatype
GET
Parent := activeParent;
END_GET
END_PROPERTY

METHOD PUBLIC SerializeWith
VAR_INPUT
	Serializer : I_Serializer;
END_VAR
Serializer.AddBool(GetBitValue());
END_METHOD

PROPERTY PUBLIC Size : UDINT
GET
Size := 1;
END_GET
END_PROPERTY

METHOD TryDeserializeFrom : BOOL
VAR_INPUT
	Deserializer : I_Deserializer;
	Feedback : I_DeserializerFeedback;
END_VAR
VAR 
	value : BOOL;
END_VAR
IF NOT Deserializer.TryGetBool(value, Feedback) THEN
	RETURN;
END_IF

SetBitValue(value);
TryDeserializeFrom := TRUE;
END_METHOD

METHOD TryMakeReferenceTo : BOOL
VAR_INPUT
	Target : I_Datatype;
END_VAR
VAR
	targetAsBit : I_BitDatatype;
END_VAR
IF NOT Target.TryResolveAsBitDatatype(targetAsBit) THEN
	RETURN;
END_IF

MakeReferenceTo(targetAsBit.Parent, targetAsBit.ByteOffset, targetAsBit.BitOffset);
TryMakeReferenceTo := TRUE;
END_METHOD

METHOD PUBLIC TryResolveAsBitDatatype : BOOL
VAR_INPUT
	Destination : REFERENCE TO I_BitDatatype;
END_VAR
Destination := this^;
TryResolveAsBitDatatype := TRUE;
END_METHOD

PROPERTY PUBLIC TypeName : T_MAXSTRING
GET
TypeName := 'BIT';
END_GET
END_PROPERTY

PROPERTY PUBLIC Value : BOOL
GET
Value := GetBitValue();
END_GET
SET
SetBitValue(Value);
END_SET
END_PROPERTY

END_FUNCTION_BLOCK

// mobject-datatypes/Primitive/_TIME_OF_DAY
{attribute 'linkalways'} 
{attribute 'no_explicit_call' := 'This FB is a CLASS and must be accessed using methods or properties'}
{attribute 'enable_dynamic_creation'}
FUNCTION_BLOCK _TIME_OF_DAY EXTENDS DatatypeBase
VAR
	localData : TIME_OF_DAY;
	activeData : REFERENCE TO TIME_OF_DAY REF= localData;
END_VAR

METHOD FB_init : BOOL
VAR_INPUT
	bInitRetains : BOOL; // if TRUE, the retain variables are initialized (warm start / cold start)
	bInCopyCode : BOOL;  // if TRUE, the instance afterwards gets moved WORDo the copy code (online change)
	InitialValue : TIME_OF_DAY;
END_VAR
localData := InitialValue;
END_METHOD

PROPERTY PUBLIC Address : PVOID
GET
Address := ADR(activeData);
END_GET
END_PROPERTY

METHOD PUBLIC ClearReference
VAR_INPUT
END_VAR
activeData REF= localData;
END_METHOD

METHOD PUBLIC Clone : I_Datatype
VAR
    pClone : POINTER TO _TIME_OF_DAY;
END_VAR
pClone := __NEW(_TIME_OF_DAY(InitialValue := Value));
Clone := pClone^;
END_METHOD

METHOD PUBLIC MakeReferenceTo
VAR_INPUT
	ReferenceTarget : REFERENCE TO TIME_OF_DAY;
END_VAR
activeData REF= ReferenceTarget;
END_METHOD

METHOD PUBLIC SerializeWith
VAR_INPUT
	Serializer : I_Serializer;
END_VAR
Serializer.AddTod(activeData);
END_METHOD

PROPERTY PUBLIC Size : UDINT
GET
Size := SIZEOF(activeData);
END_GET
END_PROPERTY

METHOD TryDeserializeFrom : BOOL
VAR_INPUT
	Deserializer : I_Deserializer;
	Feedback : I_DeserializerFeedback;
END_VAR
TryDeserializeFrom := Deserializer.TryGetTod(activeData, Feedback);
END_METHOD

METHOD TryMakeReferenceTo : BOOL
VAR_INPUT
	Target : I_Datatype;
END_VAR
VAR
	pTargetData : POINTER TO TIME_OF_DAY;
END_VAR
IF NOT (Target.TypeName = TypeName) THEN
	RETURN;
END_IF

pTargetData := Target.Address;
activeData REF= pTargetData^;
TryMakeReferenceTo := TRUE;
END_METHOD

PROPERTY PUBLIC TypeName : T_MAXSTRING
GET
TypeName := 'TIME_OF_DAY';
END_GET
END_PROPERTY

PROPERTY PUBLIC Value : REFERENCE TO TIME_OF_DAY
GET
Value REF= activeData;
END_GET
END_PROPERTY

END_FUNCTION_BLOCK

// mobject-deserialization/DeserializationFeedback/DeserializerFeedback
{attribute 'linkalways'} 
{attribute 'no_explicit_call' := 'This FB is a CLASS and must be accessed using methods or properties'}
{attribute 'enable_dynamic_creation'}
FUNCTION_BLOCK DeserializerFeedback IMPLEMENTS I_DeserializerFeedback
VAR
	errors : Stack;
	_hasError : BOOL;
	nullError : NullError;
	deserializationErrorFactory : DeserializationErrorFactory;
END_VAR

METHOD FB_exit : BOOL
VAR_INPUT
	bInCopyCode : BOOL; // if TRUE, the exit method is called for exiting an instance that is copied afterwards (online change).
END_VAR
IF bInCopyCode THEN
	RETURN;
END_IF

DisposeErrors();
END_METHOD

METHOD PRIVATE DisposeErrors : BOOL
VAR
	error : I_Error;
END_VAR
WHILE errors.TryPop(error) DO
	error.Dispose();
END_WHILE
END_METHOD

PROPERTY PUBLIC FirstError : I_Error
GET
VAR
	error : I_Error;
END_VAR
IF NOT HasError THEN
	FirstError := nullError;
	RETURN;
END_IF

IF NOT errors.TryPeek(error) THEN
	FirstError := nullError;
	RETURN;
END_IF

FirstError := error;
END_GET
END_PROPERTY

PROPERTY PUBLIC HasError : BOOL
GET
HasError := _hasError;
END_GET
END_PROPERTY

METHOD PUBLIC LogDeserializationFailedError
VAR_INPUT
	Message : T_MAXSTRING;
END_VAR
LogError(deserializationErrorFactory.CreateCustomDeserializationFailedError(Message));
END_METHOD

METHOD PUBLIC LogError
VAR_INPUT
	Error : I_Error;
END_VAR
errors.Push(Error);
_hasError := TRUE;
END_METHOD

METHOD PUBLIC LogIncorrectKeyTypeError
VAR_INPUT
	ExpectedType : T_MAXSTRING;
	ActualKey : T_MAXSTRING;
END_VAR
LogError(deserializationErrorFactory.CreateIncorrectKeyTypeError(ExpectedType, ActualKey));
END_METHOD

METHOD PUBLIC LogIncorrectTypeError
VAR_INPUT
	ExpectedType : T_MAXSTRING;
END_VAR
LogError(deserializationErrorFactory.CreateIncorrectTypeError(ExpectedType));
END_METHOD

METHOD PUBLIC LogInvalidKeyError
VAR_INPUT
END_VAR
LogError(deserializationErrorFactory.CreateInvalidKeyError());
END_METHOD

METHOD PUBLIC LogMissingKeyError
VAR_INPUT
	ExpectedKey : T_MAXSTRING;
END_VAR
LogError(deserializationErrorFactory.CreateMissingKeyError(ExpectedKey));
END_METHOD

METHOD PUBLIC Reset : BOOL
VAR_INPUT
END_VAR
DisposeErrors();
_hasError := FALSE;
END_METHOD

METHOD PUBLIC SerializeWith
VAR_INPUT
	Serializer : I_Serializer;
END_VAR
VAR
	enumerator : I_ForwardEnumerator;
	error : I_Error;
END_VAR
IF NOT HasError THEN
	RETURN;
END_IF

Serializer.AddKey('errors');
Serializer.StartArray();

enumerator := errors.GetEnumerator();

WHILE enumerator.MoveNext() DO
	IF enumerator.TryGet(error) THEN
		error.SerializeWith(Serializer);
	END_IF
END_WHILE

enumerator.Dispose();
Serializer.EndArray();
END_METHOD

END_FUNCTION_BLOCK

// mobject-errors/Errors/NullError
{attribute 'linkalways'} 
{attribute 'no_explicit_call' := 'This FB is a CLASS and must be accessed using methods or properties'}
{attribute 'enable_dynamic_creation'}
FUNCTION_BLOCK NullError EXTENDS Error
VAR
END_VAR

PROPERTY ErrorType : T_MAXSTRING
GET
END_GET
END_PROPERTY

PROPERTY PUBLIC Message : T_MAXSTRING
GET
END_GET
END_PROPERTY

METHOD PUBLIC SerializeWith
VAR_INPUT
	Serializer : I_Serializer;
END_VAR
END_METHOD

END_FUNCTION_BLOCK

// mobject-deserialization/Errors/DeserializationErrorFactory
{attribute 'linkalways'} 
{attribute 'no_explicit_call' := 'This FB is a CLASS and must be accessed using methods or properties'}
{attribute 'enable_dynamic_creation'}
FUNCTION_BLOCK DeserializationErrorFactory
VAR
END_VAR

METHOD PUBLIC CreateCustomDeserializationFailedError : I_Error
VAR_INPUT
	CustomMessage : T_MAXSTRING;
END_VAR
VAR
	pError : POINTER TO CustomDeserializationFailedError;
END_VAR
pError := __NEW(CustomDeserializationFailedError(Message := CustomMessage));
CreateCustomDeserializationFailedError := pError^;
END_METHOD

METHOD PUBLIC CreateIncorrectKeyTypeError : I_Error
VAR_INPUT
	ExpectedType : T_MAXSTRING;
	ActualKey : T_MAXSTRING;
END_VAR
VAR
	pError : POINTER TO IncorrectKeyTypeDeserializationError;
END_VAR
pError := __NEW(IncorrectKeyTypeDeserializationError(DataType := ExpectedType, Key := ActualKey));
CreateIncorrectKeyTypeError := pError^;
END_METHOD

METHOD PUBLIC CreateIncorrectTypeError : I_Error
VAR_INPUT
	ExpectedType : T_MAXSTRING;
END_VAR
VAR
	pError : POINTER TO IncorrectTypeDeserializationError;
END_VAR
pError := __NEW(IncorrectTypeDeserializationError(DataType := ExpectedType));
CreateIncorrectTypeError := pError^;
END_METHOD

METHOD PUBLIC CreateInvalidKeyError : I_Error
VAR_INPUT
END_VAR
VAR
	pError : POINTER TO InvalidKeyDeserializationError;
END_VAR
pError := __NEW(InvalidKeyDeserializationError);
CreateInvalidKeyError := pError^;
END_METHOD

METHOD PUBLIC CreateMissingKeyError : I_Error
VAR_INPUT
	ExpectedKey : T_MAXSTRING;
END_VAR
VAR
	pError : POINTER TO MissingKeyDeserializationError;
END_VAR
pError := __NEW(MissingKeyDeserializationError(Key := ExpectedKey));
CreateMissingKeyError := pError^;
END_METHOD

END_FUNCTION_BLOCK

// mobject-deserialization/Errors/CustomError/CustomDeserializationFailedError
{attribute 'linkalways'} 
{attribute 'no_explicit_call' := 'This FB is a CLASS and must be accessed using methods or properties'}
{attribute 'enable_dynamic_creation'}
FUNCTION_BLOCK CustomDeserializationFailedError EXTENDS Error
VAR
	_message : T_MAXSTRING;
END_VAR

METHOD FB_init : BOOL
VAR_INPUT
	bInitRetains : BOOL; // if TRUE, the retain variables are initialized (warm start / cold start)
	bInCopyCode : BOOL;  // if TRUE, the instance afterwards gets moved into the copy code (online change)
	Message : T_MAXSTRING;
END_VAR
this^._message := Message;
END_METHOD

PROPERTY PUBLIC ErrorType : T_MAXSTRING
GET
ErrorType := 'CUSTOM_DESERIALIZATION_ERROR';
END_GET
END_PROPERTY

PROPERTY PUBLIC Message : T_MAXSTRING
GET
Message := CONCAT('Deserialization Failed, ',_message);
END_GET
END_PROPERTY

END_FUNCTION_BLOCK

// mobject-deserialization/Errors/IncorrectType/IncorrectKeyTypeDeserializationError
{attribute 'linkalways'} 
{attribute 'no_explicit_call' := 'This FB is a CLASS and must be accessed using methods or properties'}
{attribute 'enable_dynamic_creation'}
FUNCTION_BLOCK IncorrectKeyTypeDeserializationError EXTENDS IncorrectTypeDeserializationError
VAR
	key : T_MAXSTRING;
END_VAR

METHOD FB_init : BOOL
VAR_INPUT
	bInitRetains : BOOL; // if TRUE, the retain variables are initialized (warm start / cold start)
	bInCopyCode : BOOL;  // if TRUE, the instance afterwards gets moved into the copy code (online change)
	DataType : T_MAXSTRING;
	Key : T_MAXSTRING;
END_VAR
THIS^.key := Key;
END_METHOD

PROPERTY PUBLIC Message : T_MAXSTRING
GET
VAR
	messageWithKey : T_MAXSTRING;
END_VAR
messageWithKey := concat(' for key : ',key);
Message := CONCAT(SUPER^.Message, messageWithKey);
END_GET
END_PROPERTY

END_FUNCTION_BLOCK

// mobject-deserialization/Errors/IncorrectType/IncorrectTypeDeserializationError
{attribute 'linkalways'} 
{attribute 'no_explicit_call' := 'This FB is a CLASS and must be accessed using methods or properties'}
{attribute 'enable_dynamic_creation'}
FUNCTION_BLOCK IncorrectTypeDeserializationError EXTENDS Error
VAR
	dataType : T_MAXSTRING;
END_VAR

METHOD FB_init : BOOL
VAR_INPUT
	bInitRetains : BOOL; // if TRUE, the retain variables are initialized (warm start / cold start)
	bInCopyCode : BOOL;  // if TRUE, the instance afterwards gets moved into the copy code (online change)
	DataType : T_MAXSTRING;
END_VAR
THIS^.dataType := DataType;
END_METHOD

PROPERTY PUBLIC ErrorType : T_MAXSTRING
GET
ErrorType := 'INCORRECT_DATATYPE_DESERIALIZATION_ERROR';
END_GET
END_PROPERTY

PROPERTY PUBLIC Message : T_MAXSTRING
GET
Message := CONCAT('Deserialization Failed, Incorrect Datatype : ', dataType);
END_GET
END_PROPERTY

END_FUNCTION_BLOCK

// mobject-deserialization/Errors/Invalid Key/InvalidKeyDeserializationError
{attribute 'linkalways'} 
{attribute 'no_explicit_call' := 'This FB is a CLASS and must be accessed using methods or properties'}
{attribute 'enable_dynamic_creation'}
FUNCTION_BLOCK InvalidKeyDeserializationError EXTENDS Error
VAR
END_VAR

PROPERTY PUBLIC ErrorType : T_MAXSTRING
GET
ErrorType := 'INVALID_KEY_DESERIALIZATION_ERROR';
END_GET
END_PROPERTY

PROPERTY PUBLIC Message : T_MAXSTRING
GET
Message := 'Deserialization Failed, Key Cannot Be Empty';
END_GET
END_PROPERTY

END_FUNCTION_BLOCK

// mobject-deserialization/Errors/Missing Key/MissingKeyDeserializationError
{attribute 'linkalways'} 
{attribute 'no_explicit_call' := 'This FB is a CLASS and must be accessed using methods or properties'}
{attribute 'enable_dynamic_creation'}
FUNCTION_BLOCK MissingKeyDeserializationError EXTENDS Error
VAR
	key : T_MAXSTRING;
END_VAR

METHOD FB_init : BOOL
VAR_INPUT
	bInitRetains : BOOL; // if TRUE, the retain variables are initialized (warm start / cold start)
	bInCopyCode : BOOL;  // if TRUE, the instance afterwards gets moved into the copy code (online change)
	Key : T_MAXSTRING;
END_VAR
this^.key := Key;
END_METHOD

PROPERTY PUBLIC ErrorType : T_MAXSTRING
GET
ErrorType := 'MISSING_KEY_DESERIALIZATION_ERROR';
END_GET
END_PROPERTY

PROPERTY PUBLIC Message : T_MAXSTRING
GET
Message := CONCAT('Deserialization Failed, Missing Key : ',key);
END_GET
END_PROPERTY

END_FUNCTION_BLOCK

// mobject-deserialization/GarbageCollector/DeserializerGarbageCollector
{attribute 'linkalways'} 
{attribute 'no_explicit_call' := 'This FB is a CLASS and must be accessed using methods or properties'}
{attribute 'enable_dynamic_creation'}
FUNCTION_BLOCK DeserializerGarbageCollector EXTENDS Disposable Implements I_DeserializerGarbageCollector
VAR
	deserializers : Stack;
END_VAR

METHOD FB_exit : BOOL
VAR_INPUT
	bInCopyCode : BOOL; // if TRUE, the exit method is called for exiting an instance that is copied afterwards (online change).
END_VAR
IF bInCopyCode THEN
	RETURN;
END_IF

DisposeAll();
END_METHOD

METHOD PROTECTED DisposeAll
VAR
	deserializer : I_Deserializer;
END_VAR
WHILE deserializers.TryPop(deserializer) DO
	deserializer.Dispose();
END_WHILE
END_METHOD

METHOD PUBLIC Deregister
VAR_INPUT
	Deserializer : I_Deserializer;
END_VAR
deserializers.TryRemoveItem(Deserializer);
END_METHOD

METHOD PUBLIC Execute
VAR_INPUT
END_VAR
DisposeAll();
END_METHOD

METHOD PUBLIC Register
VAR_INPUT
	Deserializer : I_Deserializer;
END_VAR
deserializers.Push(Deserializer);
END_METHOD

END_FUNCTION_BLOCK

// mobject-deserialization/GarbageCollector/I_DeserializerGarbageCollector
INTERFACE I_DeserializerGarbageCollector EXTENDS __SYSTEM.IQueryInterface

METHOD PUBLIC Deregister
VAR_INPUT
	Deserializer : I_Deserializer;
END_VAR
END_METHOD

METHOD PUBLIC Register
VAR_INPUT
	Deserializer : I_Deserializer;
END_VAR
END_METHOD

END_INTERFACE

// mobject-json/_Internal/Events/JsonDeserializerChangedEvent
{attribute 'linkalways'} 
{attribute 'no_explicit_call' := 'This FB is a CLASS and must be accessed using methods or properties'}
{attribute 'enable_dynamic_creation'}
FUNCTION_BLOCK JsonDeserializerChangedEvent EXTENDS JsonDeserializerEvent IMPLEMENTS I_JsonDeserializerChangedEvent

END_FUNCTION_BLOCK

// mobject-json/_Internal/Events/JsonDeserializerEvent
{attribute 'linkalways'} 
{attribute 'no_explicit_call' := 'This FB is a CLASS and must be accessed using methods or properties'}
{attribute 'enable_dynamic_creation'}
FUNCTION_BLOCK ABSTRACT JsonDeserializerEvent EXTENDS Disposable
VAR
	_target : I_JsonDeserializer;
END_VAR

METHOD FB_init : BOOL
VAR_INPUT
	bInitRetains : BOOL; // if TRUE, the retain variables are initialized (warm start / cold start)
	bInCopyCode : BOOL;  // if TRUE, the instance afterwards gets moved into the copy code (online change)
	Target : I_JsonDeserializer;
END_VAR
This^._target := Target;
END_METHOD

PROPERTY PUBLIC Target : I_JsonDeserializer
GET
PUBLIC
Target := _target;
END_GET
END_PROPERTY

END_FUNCTION_BLOCK

// mobject-json/JsonDeserializer/I_JsonDeserializer
INTERFACE I_JsonDeserializer EXTENDS I_Deserializer, I_EventEmitter, I_Disposable

END_INTERFACE

// mobject-json/JsonDeserializer/Events/I_JsonDeserializerChangedEvent
INTERFACE I_JsonDeserializerChangedEvent EXTENDS I_Event

PROPERTY PUBLIC Target : I_JsonDeserializer
GET
END_GET
END_PROPERTY

END_INTERFACE

// mobject-json/_Internal/Events/JsonDeserializerDisposedEvent
{attribute 'linkalways'} 
{attribute 'no_explicit_call' := 'This FB is a CLASS and must be accessed using methods or properties'}
{attribute 'enable_dynamic_creation'}
FUNCTION_BLOCK JsonDeserializerDisposedEvent EXTENDS JsonDeserializerEvent IMPLEMENTS I_JsonDeserializerDisposedEvent

END_FUNCTION_BLOCK

// mobject-json/JsonDeserializer/Events/I_JsonDeserializerDisposedEvent
INTERFACE I_JsonDeserializerDisposedEvent EXTENDS I_Event

PROPERTY PUBLIC Target : I_JsonDeserializer
GET
END_GET
END_PROPERTY

END_INTERFACE

// mobject-json/_Internal/JsonDeserializerForwardEnumerator/JsonDeserializerArrayForwardEnumerator
{attribute 'linkalways'} 
{attribute 'no_explicit_call' := 'This FB is a CLASS and must be accessed using methods or properties'}
{attribute 'enable_dynamic_creation'}
FUNCTION_BLOCK JsonDeserializerArrayForwardEnumerator EXTENDS Disposable IMPLEMENTS I_DeserializerArrayForwardEnumerator, I_EventHandler
VAR
	parent : I_JsonDeserializer;
	jsonParser : REFERENCE TO JsonDomParser;
	root : SJsonValue;
	garbageCollector : I_DeserializerGarbageCollector;
	nullNode : I_Deserializer;
	moveNextCalled : BOOL := FALSE;
	invalid : BOOL := FALSE; 
	nextArrayPosition : SJsonValue;
	arrayBeginPosition : SJsonValue;
	arrayEndPosition : SJsonValue;
	currentDeserializer : I_Deserializer;
	_index : DINT;
END_VAR

METHOD FB_init : BOOL
VAR_INPUT
	bInitRetains : BOOL; // if TRUE, the retain variables are initialized (warm start / cold start)
	bInCopyCode : BOOL;  // if TRUE, the instance afterwards gets moved into the copy code (online change)
	ParentJsonDeserializer : I_JsonDeserializer;
	ParentJsonDomParser : REFERENCE TO JsonDomParser;
	NodeRoot : SJsonValue;
	ParentGarbageCollector : I_DeserializerGarbageCollector;
	ParentNullDeserializer : I_Deserializer;
END_VAR
THIS^.parent := ParentJsonDeserializer;
THIS^.jsonParser REF= ParentJsonDomParser;
THIS^.root := NodeRoot;
THIS^.garbageCollector := ParentGarbageCollector;
THIS^.nullNode := ParentNullDeserializer;

Initialize();

Parent.OnEvent('OnChanged',THIS^);
Parent.OnEvent('OnDisposed',THIS^);
END_METHOD

METHOD FB_exit : BOOL
VAR_INPUT
	bInCopyCode : BOOL; // if TRUE, the exit method is called for exiting an instance that is copied afterwards (online change).
END_VAR
IF bInCopyCode THEN
	RETURN;
END_IF

IF parent = 0 THEN
	RETURN;
END_IF

parent.OffEvent('OnChanged',THIS^);
parent.OffEvent('OnDisposed',THIS^);
END_METHOD

METHOD PROTECTED CreateDeserializer : I_Deserializer
VAR_INPUT
	DeserializerRoot : SJsonValue;
END_VAR
VAR 
	pNode : POINTER TO JsonDeserializerNode;
END_VAR
pNode := __NEW(JsonDeserializerNode(
	ParentJsonDeserializer := parent,
	ParentJsonDomParser := jsonParser, 
	NodeRoot := DeserializerRoot, 
	ParentGarbageCollector := garbageCollector, 
	ParentNullDeserializer := nullNode
));

CreateDeserializer := pNode^;
END_METHOD

METHOD PROTECTED Initialize
VAR_INPUT
END_VAR
IF NOT jsonParser.IsArray(root) THEN
	invalid := TRUE;
	RETURN;
END_IF

arrayBeginPosition := jsonParser.ArrayBegin(root);
arrayEndPosition := jsonParser.ArrayEnd(root);

IF arrayBeginPosition = 0 THEN
	invalid := TRUE;
	RETURN;
END_IF

IF arrayEndPosition = 0 THEN
	invalid := TRUE;
	RETURN;
END_IF
END_METHOD

METHOD PROTECTED UpdateCurrentDeserializer
VAR_INPUT
	Root : SJsonValue;
END_VAR
VAR
	newRoot : SJsonValue;
END_VAR
IF currentDeserializer <> 0 THEN
	currentDeserializer.Dispose();
	currentDeserializer := 0;
END_IF

IF invalid THEN
	RETURN;
END_IF

newRoot := jsonParser.GetArrayValue(Root);

IF newRoot = 0 THEN
	RETURN;
END_IF

currentDeserializer := CreateDeserializer(newRoot);
END_METHOD

PROPERTY PUBLIC Current : I_Deserializer
GET
IF NOT IsValid THEN
	Current := nullNode;
	RETURN;
END_IF

IF currentDeserializer = 0 THEN
	Current := nullNode;
	RETURN;
END_IF

Current := currentDeserializer;
END_GET
END_PROPERTY

METHOD PUBLIC HandleEvent
VAR_INPUT
	Event : I_Event;
END_VAR
VAR
	changedEvent : I_JsonDeserializerChangedEvent;
	disposedEvent : I_JsonDeserializerDisposedEvent;
END_VAR
IF __QUERYINTERFACE(Event, changedEvent) THEN
	invalid := TRUE;
ELSIF __QUERYINTERFACE(Event, disposedEvent) THEN
	parent := 0;
	Dispose();
END_IF
END_METHOD

PROPERTY Index : DINT
GET
Index := _index;
END_GET
END_PROPERTY

PROPERTY PUBLIC IsValid : BOOL
GET
PUBLIC
IF invalid THEN
	RETURN;
END_IF

IF parent = 0 THEN
	RETURN;
END_IF

IsValid := TRUE;
END_GET
END_PROPERTY

METHOD PUBLIC MoveNext : BOOL
IF invalid THEN
    RETURN;
END_IF

// Handle the initial move
IF NOT moveNextCalled THEN
    moveNextCalled := TRUE;
    UpdateCurrentDeserializer(arrayBeginPosition);
	nextArrayPosition := jsonParser.NextArray(arrayBeginPosition);
	_index := _index + 1;
	MoveNext := TRUE;
    RETURN;
END_IF

// Handle subsequent moves
IF nextArrayPosition <> arrayEndPosition THEN
	UpdateCurrentDeserializer(nextArrayPosition);
	nextArrayPosition := jsonParser.NextArray(nextArrayPosition);
	_index := _index + 1;
	MoveNext := TRUE;
END_IF
END_METHOD

END_FUNCTION_BLOCK

// mobject-json/JsonDomParser/JsonDomParser
{attribute 'linkalways'} 
{attribute 'no_explicit_call' := 'This FB is a CLASS and must be accessed using methods or properties'}
{attribute 'enable_dynamic_creation'}
FUNCTION_BLOCK JsonDomParser EXTENDS FB_JsonDynDomParser
VAR
	currentlyParsingType : (NOTHING, DOT_NOTATION_PROPERTY, BRACKET_NOTATION_PROPERTY_OR_ARRAY, BRACKET_NOTATION_PROPERTY_ELEMENT, BRACKET_NOTATION_ARRAY_ELEMENT);
	readWriteDataType : FB_JsonReadWriteDataType;
END_VAR

METHOD PRIVATE TrySetBool : BOOL
VAR_INPUT
	JsonValue : SJsonValue;
	Source : ANY;
END_VAR
VAR
	_BOOL : BOOL;
END_VAR
IF Source.TypeClass <> __SYSTEM.TYPE_CLASS.TYPE_BOOL THEN	
	RETURN;
END_IF

memcpy(ADR(_BOOL),Source.pValue,DINT_TO_UDINT(Source.diSize));
SetBool(jsonValue,_BOOL);
TrySetBool := TRUE;
END_METHOD

METHOD PRIVATE TrySetDouble : BOOL
VAR_INPUT
	JsonValue : SJsonValue;
	Source : ANY;
END_VAR
VAR
	convertSuccessful : BOOL;
	_REAL : REAL;
	_LREAL : LREAL;
END_VAR
CASE Source.TypeClass OF 

	__SYSTEM.TYPE_CLASS.TYPE_REAL : 
		memcpy(ADR(_REAL),Source.pValue,DINT_TO_UDINT(Source.diSize));
		convertSuccessful := TryConvert_Source_TO_Destination(_REAL,_LREAL);
	
	__SYSTEM.TYPE_CLASS.TYPE_LREAL : 
		memcpy(ADR(_LREAL),Source.pValue,DINT_TO_UDINT(Source.diSize));
		convertSuccessful := TRUE;
		
ELSE 
		
	RETURN;
		
END_CASE

IF NOT convertSuccessful THEN
	RETURN;
END_IF

SetDouble(jsonValue,_LREAL);
TrySetDouble := TRUE;
END_METHOD

METHOD PRIVATE TrySetInt : BOOL
VAR_INPUT
	JsonValue : SJsonValue;
	Source : ANY;
END_VAR
VAR
	convertSuccessful : BOOL;
	_SINT : USINT;	
	_INT : UINT;
	_DINT : DINT;
END_VAR
CASE Source.TypeClass OF
		
	__SYSTEM.TYPE_CLASS.TYPE_SINT : 
		memcpy(ADR(_SINT),Source.pValue,DINT_TO_UDINT(Source.diSize));
		convertSuccessful := TryConvert_Source_TO_Destination(_SINT,_DINT);
		
	__SYSTEM.TYPE_CLASS.TYPE_INT : 
		memcpy(ADR(_INT),Source.pValue,DINT_TO_UDINT(Source.diSize));
		convertSuccessful := TryConvert_Source_TO_Destination(_INT,_DINT);
		
	__SYSTEM.TYPE_CLASS.TYPE_DINT : 
		memcpy(ADR(_DINT),Source.pValue,DINT_TO_UDINT(Source.diSize));
		convertSuccessful := TRUE;
		
ELSE 
		
	RETURN;
		
END_CASE

IF NOT convertSuccessful THEN
	RETURN;
END_IF

SetInt(jsonValue,_DINT); // Not a typo, SetInt actually takes a DINT
TrySetInt := TRUE;
END_METHOD

METHOD PRIVATE TrySetInt64 : BOOL
VAR_INPUT
	JsonValue : SJsonValue;
	Source : ANY;
END_VAR
VAR
	_LINT : LINT;
END_VAR
IF Source.TypeClass <> __SYSTEM.TYPE_CLASS.TYPE_LINT THEN	
	RETURN;
END_IF

memcpy(ADR(_LINT),Source.pValue,DINT_TO_UDINT(Source.diSize));
SetInt64(jsonValue,_LINT);
TrySetInt64 := TRUE;
END_METHOD

METHOD PRIVATE TrySetString : BOOL
VAR_INPUT
	JsonValue : SJsonValue;
	Source : ANY;
END_VAR
VAR
	_STRING : POINTER TO STRING(1);
END_VAR
IF Source.TypeClass <> __SYSTEM.TYPE_CLASS.TYPE_STRING THEN	
	RETURN;
END_IF

_STRING := Source.pValue;

SetString(jsonValue,_STRING^);
TrySetString := TRUE;
END_METHOD

METHOD PRIVATE TrySetUint : BOOL
VAR_INPUT
	JsonValue : SJsonValue;
	Source : ANY;
END_VAR
VAR
	convertSuccessful : BOOL;
	_BYTE : BYTE;
	_WORD : WORD;
	_DWORD : DWORD;	
	_USINT : USINT;	
	_UINT : UINT;
	_UDINT : UDINT;
END_VAR
CASE Source.TypeClass OF 

	__SYSTEM.TYPE_CLASS.TYPE_BYTE : 
		memcpy(ADR(_BYTE),Source.pValue,DINT_TO_UDINT(Source.diSize));
		convertSuccessful := TryConvert_Source_TO_Destination(_BYTE,_UDINT);
	
	__SYSTEM.TYPE_CLASS.TYPE_WORD : 
		memcpy(ADR(_WORD),Source.pValue,DINT_TO_UDINT(Source.diSize));
		convertSuccessful := TryConvert_Source_TO_Destination(_WORD,_UDINT);
		
	__SYSTEM.TYPE_CLASS.TYPE_DWORD : 
		memcpy(ADR(_DWORD),Source.pValue,DINT_TO_UDINT(Source.diSize));
		convertSuccessful := TryConvert_Source_TO_Destination(_DWORD,_UDINT);
		
	__SYSTEM.TYPE_CLASS.TYPE_USINT : 
		memcpy(ADR(_USINT),Source.pValue,DINT_TO_UDINT(Source.diSize));
		convertSuccessful := TryConvert_Source_TO_Destination(_USINT,_UDINT);
		
	__SYSTEM.TYPE_CLASS.TYPE_UINT : 
		memcpy(ADR(_UINT),Source.pValue,DINT_TO_UDINT(Source.diSize));
		convertSuccessful := TryConvert_Source_TO_Destination(_UINT,_UDINT);
		
	__SYSTEM.TYPE_CLASS.TYPE_UDINT : 
		memcpy(ADR(_UDINT),Source.pValue,DINT_TO_UDINT(Source.diSize));
		convertSuccessful := TRUE;
		
ELSE 
		
	RETURN;
		
END_CASE

IF NOT convertSuccessful THEN
	RETURN;
END_IF

SetUint(jsonValue,_UDINT); // Not a typo, SetUnit actually takes a UDINT
TrySetUint := TRUE;
END_METHOD

METHOD PRIVATE TrySetUint64 : BOOL
VAR_INPUT
	JsonValue : SJsonValue;
	Source : ANY;
END_VAR
VAR
	convertSuccessful : BOOL;
	_LWORD : LWORD;
	_ULINT : ULINT;
END_VAR
CASE Source.TypeClass OF 

	__SYSTEM.TYPE_CLASS.TYPE_LWORD : 
		memcpy(ADR(_LWORD),Source.pValue,DINT_TO_UDINT(Source.diSize));
		convertSuccessful := TryConvert_Source_TO_Destination(_LWORD,_ULINT);
	
	__SYSTEM.TYPE_CLASS.TYPE_ULINT : 
		memcpy(ADR(_ULINT),Source.pValue,DINT_TO_UDINT(Source.diSize));
		convertSuccessful := TRUE;
		
ELSE 
		
	RETURN;
		
END_CASE

IF NOT convertSuccessful THEN
	RETURN;
END_IF

SetUint64(jsonValue,_ULINT);
TrySetUint64 := TRUE;
END_METHOD

METHOD PUBLIC TryLocate : BOOL
VAR_INPUT
	Path : T_MaxString;
	Destination : REFERENCE TO SJsonValue;
END_VAR
VAR
	jsonDomNavigator : JsonDomNavigator(THIS^);
	jsonPathSyntaxParser : JsonPathSyntaxParser;
	jsonValue : SJsonValue;
END_VAR
jsonPathSyntaxParser.Parse(Path, jsonDomNavigator);
jsonValue := jsonDomNavigator.CurrentNode;

IF jsonValue = 0 THEN
	RETURN;
END_IF

Destination := jsonValue;
TryLocate := TRUE;
END_METHOD

METHOD PUBLIC TryModify : BOOL
VAR_INPUT
	Path : T_MaxString;
	Source : ANY;
END_VAR
VAR
	jsonDomNavigator : JsonDomNavigator(THIS^);
	jsonPathSyntaxParser : JsonPathSyntaxParser;
	jsonValue : SJsonValue;
END_VAR
jsonPathSyntaxParser.Parse(Path, jsonDomNavigator);
jsonValue := jsonDomNavigator.CurrentNode;

IF jsonValue = 0 THEN
	RETURN;
END_IF

IF IsObject(jsonValue) THEN
	RETURN;
END_IF

IF TrySetBool(jsonValue, Source) THEN
	TryModify := TRUE;
	RETURN;
END_IF

IF TrySetString(jsonValue, Source) THEN
	TryModify := TRUE;
	RETURN;
END_IF

IF TrySetInt(jsonValue, Source) THEN
	TryModify := TRUE;
	RETURN;
END_IF

IF TrySetUint(jsonValue, Source) THEN
	TryModify := TRUE;
	RETURN;
END_IF

IF TrySetDouble(jsonValue, Source) THEN
	TryModify := TRUE;
	RETURN;
END_IF

IF TrySetInt64(jsonValue, Source) THEN
	TryModify := TRUE;
	RETURN;
END_IF

IF TrySetUint64(jsonValue, Source) THEN
	TryModify := TRUE;
	RETURN;
END_IF
END_METHOD

METHOD PUBLIC TryRead : BOOL
VAR_INPUT
	Path : T_MaxString;
	Destination : ANY;
END_VAR
VAR
	jsonDomNavigator : JsonDomNavigator(THIS^);
	jsonPathSyntaxParser : JsonPathSyntaxParser;
	jsonValue : SJsonValue;
	_BOOL : BOOL;
	_DINT : DINT;
	_LINT : LINT;
	_UDINT : UDINT;
	_ULINT : ULINT;
	_LREAL : LREAL;
	_STRING : POINTER TO STRING(1);
END_VAR
jsonPathSyntaxParser.Parse(Path, jsonDomNavigator);
jsonValue := jsonDomNavigator.CurrentNode;

IF jsonValue = 0 THEN
	RETURN;
END_IF

IF IsBool(jsonValue) THEN
	_BOOL := GetBool(jsonValue);
	TryRead := TryConvert_BOOL_TO_DESTINATION(_BOOL,Destination);
	RETURN;
END_IF

IF IsInt(jsonValue) THEN
	_DINT := GetInt(jsonValue);
	TryRead := TryConvert_DINT_TO_DESTINATION(_DINT,Destination);
	RETURN;
END_IF

IF IsInt64(jsonValue) THEN
	_LINT := GetInt64(jsonValue);
	TryRead := TryConvert_LINT_TO_DESTINATION(_LINT,Destination);
	RETURN;
END_IF

IF IsUInt(jsonValue) THEN
	_UDINT := GetUInt(jsonValue);
	TryRead := TryConvert_UDINT_TO_DESTINATION(_UDINT,Destination);
	RETURN;
END_IF

IF IsUInt64(jsonValue) THEN
	_ULINT := GetUInt64(jsonValue);
	TryRead := TryConvert_ULINT_TO_DESTINATION(_ULINT,Destination);
	RETURN;
END_IF

IF IsDouble(jsonValue) THEN
	_LREAL := GetDouble(jsonValue);
	TryRead := TryConvert_LREAL_TO_DESTINATION(_LREAL,Destination);
	RETURN;
END_IF

IF IsString(jsonValue) AND Destination.TypeClass = __SYSTEM.TYPE_CLASS.TYPE_STRING THEN
	_STRING := Destination.pValue;
	IF (CopyString(jsonValue,_STRING^,DINT_TO_UDINT(Destination.diSize)) > 0) THEN;
		TryRead := TRUE;
		RETURN;
	END_IF
END_IF
END_METHOD

METHOD PUBLIC TryWrite : BOOL
VAR_INPUT
	Path : T_MaxString;
	Source : ANY;
END_VAR
VAR
	jsonDomCreator : JsonDomCreator(THIS^);
	jsonPathSyntaxParser : JsonPathSyntaxParser;
	jsonValue : SJsonValue;
END_VAR
jsonPathSyntaxParser.Parse(Path, jsonDomCreator);
jsonValue := jsonDomCreator.CurrentNode;

IF jsonValue = 0 THEN
	RETURN;
END_IF

IF IsObject(jsonValue) THEN
	RETURN;
END_IF

IF TrySetBool(jsonValue, Source) THEN
	TryWrite := TRUE;
	RETURN;
END_IF

IF TrySetString(jsonValue, Source) THEN
	TryWrite := TRUE;
	RETURN;
END_IF

IF TrySetInt(jsonValue, Source) THEN
	TryWrite := TRUE;
	RETURN;
END_IF

IF TrySetUint(jsonValue, Source) THEN
	TryWrite := TRUE;
	RETURN;
END_IF

IF TrySetDouble(jsonValue, Source) THEN
	TryWrite := TRUE;
	RETURN;
END_IF

IF TrySetInt64(jsonValue, Source) THEN
	TryWrite := TRUE;
	RETURN;
END_IF

IF TrySetUint64(jsonValue, Source) THEN
	TryWrite := TRUE;
	RETURN;
END_IF
END_METHOD

END_FUNCTION_BLOCK

// mobject-json/_Internal/JsonPathSyntaxParser/JsonPathSyntaxParser
{attribute 'linkalways'} 
{attribute 'no_explicit_call' := 'This FB is a CLASS and must be accessed using methods or properties'}
{attribute 'enable_dynamic_creation'}
FUNCTION_BLOCK JsonPathSyntaxParser
VAR
	currentlyParsingType : (NOTHING, DOT_NOTATION_PROPERTY, BRACKET_NOTATION_PROPERTY_OR_ARRAY, BRACKET_NOTATION_PROPERTY_ELEMENT, BRACKET_NOTATION_ARRAY_ELEMENT);
END_VAR

METHOD PUBLIC Parse
VAR_INPUT
	Path : REFERENCE TO STRING;
	JsonPathVisitor : I_JsonPathVisitor;
END_VAR
VAR
	currentCharacterPositionInPath : UDINT;
	currentElementStart : UDINT;
	currentElementEnd : UDINT;
	currentElementLength : UDINT;
	elementText : T_MAXSTRING;
	endOfRepeat : BOOL;
END_VAR
VAR CONSTANT
	PERIOD : BYTE := 16#2E; // .
	DOLLAR_SIGN : BYTE := 16#24; // $
	SINGLE_QUOTE : BYTE := 16#27; // '
	LEFT_SQUARE_BRACKET : BYTE := 16#5B; // [
	RIGHT_SQUARE_BRACKET : BYTE := 16#5D; // ]
	NULL : BYTE := 0; // null
END_VAR
JsonPathVisitor.StartOfParse();

IF Path[0] = NULL THEN
	JsonPathVisitor.EndOfParse();
	RETURN;
END_IF

currentCharacterPositionInPath := 0;
currentlyParsingType := NOTHING;

REPEAT 
	
	IF Path[currentCharacterPositionInPath] = NULL THEN
		 endOfRepeat := TRUE;
	END_IF
		
	CASE currentlyParsingType OF
		
		NOTHING: 
		
